(* CODESYS project plc_chalet_xplanar.library
   Title: CHALET_XPlanar
   Version: 4.3.3
   Placeholder: CHALET_XPlanar
   Company: Beckhoff CH

Project tree, tasks and I/O mapping:
  libraries: CHALET_BaseComponents, * (Beckhoff CH); CHALET_Nc, * (Beckhoff CH); Tc2_EtherCAT, * (Beckhoff Automation GmbH); Tc2_Math, * (Beckhoff Automation GmbH); Tc2_Standard, * (Beckhoff Automation GmbH); Tc2_System, * (Beckhoff Automation GmbH); Tc2_Utilities, * (Beckhoff Automation GmbH); Tc3_EventLogger, * (Beckhoff Automation GmbH); Tc3_Mc3Definitions, * (Beckhoff Automation GmbH); Tc3_Mc3PlanarMotion, * (Beckhoff Automation GmbH); Tc3_Module, * (Beckhoff Automation GmbH); Tc3_Physics, * (Beckhoff Automation GmbH); Tc3_XPlanarUtility, * (Beckhoff Automation GmbH & Co. KG)
  COMPONENTs/
    Environment/
      function block FB_XP_Environment [ST]: AddToGroup, RemoveFromGroup, Clear, Configure, FB_init, Feedback, Initialize, Mapped, OID, PlanarEnvironment, Update, UtilityEnvirement
      interface I_XP_Environment: AddToGroup, Clear, Configure, Feedback, Initialize, Mapped, OID, PlanarEnvironment, RemoveFromGroup, Update, UtilityEnvirement
    Feedback/
      function block FB_XP_Feedback [ST]: ClearObjectInfo, ObjectInfo
      interface I_XP_Feedback: ObjectInfo
    Group/
      function block FB_XP_Group [ST]: AddEnvironment, AddMover, AddTrack, Disable, Enable, FB_init, Feedback, Initialize, Mapped, OID, PlanarGroup, Reset, Update
      interface I_XP_Group: AddEnvironment, AddMover, AddTrack, Disable, Enable, Feedback, Initialize, Mapped, OID, PlanarGroup, Reset, Update
    Mover/
      ProductData/
        function block FB_XP_ProductData [ST]: LinkedMover, LinkToMover
        interface I_XP_ProductData: LinkedMover, LinkToMover
      function block FB_XP_Mover [ST]: DynConstraint, SetDynConstraint_A, SetDynConstraint_B, SetDynConstraint_C, SetDynConstraint_Path, SetDynConstraint_X, SetDynConstraint_Y, SetDynConstraint_Z, AxisExtSetpointA, AxisExtSetpointB, AxisExtSetpointC, AxisExtSetpointX, AxisExtSetpointY, AxisExtSetpointZ, StartExternalSetpoint, StopExternalSetpoint, UpdateExternalSetpoint, AddToGroup, RemoveFromGroup, Halt, MoveA, MoveB, MoveC, MoveXY, MoveZ, Disable, Enable, Reset, CommandMode, LagDistanceXY, PositionAct, PositionSet, CurrentTrack, DistToTrack, JoinTrack, LastCmdTargedGap, LastCmdTargedPosition, LastCmdTargedTrack, MoveOnTrack, MoveOnTrack_ShortestWay, MoveOnTrackToStation, ParentStation, PositionOnTrack, TargetStation, TcIoXPlanarMover, UtilityMover, DistToParentStation, FB_init, Feedback, Initialize, Mapped, Mode, OID, PlanarMover, Prepare, ProductData, Route, Update
      interface I_XP_Mover: AddToGroup, RemoveFromGroup, Halt, MoveA, MoveB, MoveC, MoveXY, MoveZ, Disable, Enable, Reset, CurrentTrack, DistToTrack, JoinTrack, LastCmdTargedGap, LastCmdTargedPosition, LastCmdTargedTrack, MoveOnTrack, MoveOnTrack_ShortestWay, MoveOnTrackToStation, ParentStation, PositionOnTrack, TargetStation, TcIoXPlanarMover, UtilityMover, DistToParentStation, Feedback, Mapped, Mode, OID, PlanarMover, Route
      interface I_XP_Mover_PLC: DynConstraint, SetDynConstraint_A, SetDynConstraint_B, SetDynConstraint_C, SetDynConstraint_Path, SetDynConstraint_X, SetDynConstraint_Y, SetDynConstraint_Z, AxisExtSetpointA, AxisExtSetpointB, AxisExtSetpointC, AxisExtSetpointX, AxisExtSetpointY, AxisExtSetpointZ, StartExternalSetpoint, StopExternalSetpoint, Halt, MoveA, MoveB, MoveC, MoveXY, MoveZ, CommandMode, LagDistanceXY, PositionAct, PositionSet, CurrentTrack, LastCmdTargedGap, LastCmdTargedPosition, LastCmdTargedTrack, ParentStation, PositionOnTrack, TargetStation, TcIoXPlanarMover, UtilityMover, DistToParentStation, Feedback, LUID, Mapped, OID, PlanarMover, ProductData
    Optional/
      Casting/
        function ToXpMover [ST]
        function ToXpStation [ST]
        function ToXpTrack [ST]
      Trigger/
        function block FB_XP_Trigger [ST]: AccocietedTrack, FB_init, HR, Initialize, ListOfMoversToCheck, MoverAtTrigger, MoverDetected, PositionOnTrack, Prepare, TimeStamp, TriggerDirection, Update
        interface I_XP_Trigger: AccocietedTrack, HR, ListOfMoversToCheck, MoverAtTrigger, MoverDetected, PositionOnTrack, TimeStamp, TriggerDirection
      Zone/
        function block FB_XP_SoretedListOfMover [ST]: CtsMoversInZone, FB_init, Initialize, MoversInZone, Prepare, Update
        interface I_XP_Zone: CtsMoversInZone, MoversInZone
      function F_GetDistToPosModulo [ST]
      function F_InLimitTest [ST]
      function block FB_XP_Path [ST]: DistanceToDestiantion, Length, LUID, PointerToThis, StationDestination, StationStart, TracksUsed
      interface I_XP_Path: DistanceToDestiantion, Length, PointerToThis, StationDestination, StationStart, TracksUsed
    Stationen/
      function block FB_XP_Station [ST]: CheckInvalideParameter, GetAccocietedTrack, GetDecisionDistance, GetPathsAhead, GetPathsBehind, GetPosOnTrack, GetStationAhead, GetStationBehinde, SetTrackObjName, Configure, CtsEmptySpaceInQueue, CtsMoversInQueue, MoverQueueSize, MoversInPlace, MoversInQueue, ReadyToRecvMovers, SendMoversToStation, SuppressDynamicsChange, TargetGroupe, TargetPosMonitoringTime, TargetPosWindow, ProcessSimulationActive, Simulation, SimulationMode, AccocietedTrack, AddMoverToQueue, AssignedMovers, DeleteMoversQueue, FB_exit, FB_init, Feedback, Filter, Initialize, MoverGapAtExit, MoverVelocityAtExit, OID, PathsAhead, PathsBehinde, PositionOnTrack, PositionOnTrackXY, PositionXY, Prepare, SearchNextBestStationByName, StationsAhead, StationsBehinde, Update
      interface I_XP_Station: AccocietedTrack, AddMoverToQueue, AssignedMovers, Configure, CtsEmptySpaceInQueue, DeleteMoversQueue, Filter, PathsAhead, PathsBehinde, PositionOnTrack, PositionOnTrackXY, PositionXY, ReadyToRecvMovers, SearchNextBestStationByName, SendMoversToStation, StationsAhead, StationsBehinde, TargetGroupe, Update
      interface I_XP_Station_PLC: CtsEmptySpaceInQueue, CtsMoversInQueue, LUID, MoverQueueSize, MoversInPlace, MoversInQueue, ReadyToRecvMovers, SendMoversToStation, TargetPosMonitoringTime, TargetPosWindow, ProcessSimulationActive, SimulationMode, AccocietedTrack, Feedback, Filter, MoverGapAtExit, PositionOnTrack, PositionOnTrackXY, PositionXY, StationsAhead, StationsBehinde, TargetGroupe
      data type ST_PathFinder_1
    System/
      function block FB_XP_System [ST]: JoiningStation, JoiningTrack, Disable, Disabled, Disabling, Enable, Enabled, Enabling, Initialize, Initialized, CheckTargetExists, Station, LinkEnvironment, LinkGroup, RegisterMover, RegisterStation, RegisterTrack, RegisterTrigger, RegisterZone, Enviroment, FB_init, Feedback, Movers, Stations, Tracks, Triggers, Update, XPlanarTaskAdsPort, Zones
      interface I_XP_System_PLC: CheckTargetExists, Disable, Disabled, Enable, Enabled, Enviroment, Feedback, Initialize, Initialized, Movers, Station, Stations, Tracks, Triggers, Update, Zones
      interface I_XP_System_Registration: LinkEnvironment, LinkGroup, RegisterMover, RegisterStation, RegisterTrack, RegisterTrigger, RegisterZone, Disabled, Enabled, Enviroment, Movers, Stations, Tracks, Triggers, XPlanarTaskAdsPort, Zones
    Track/
      function block FB_XP_Track [ST]: Configure, Configuring, Disable, Enable, AddToGroup, RemoveFromGroup, AddMover, ClosedLoop, CtsMoversOnTrack, FB_init, Feedback, Initialize, Length, Mapped, OID, PlanarTrack, Prepare, Reset, StationsOnTrack, TracksAhead, TracksBehinde, TracksEndAtThis, TracksStartFromThis, Update
      interface I_XP_Track: AddMover, AddToGroup, ClosedLoop, Configure, Configuring, CtsMoversOnTrack, Disable, Enable, Feedback, Length, OID, PlanarTrack, RemoveFromGroup, Reset, StationsOnTrack, TracksAhead, TracksBehinde, TracksEndAtThis, TracksStartFromThis
      interface I_XP_Track_PLC: CtsMoversOnTrack, Feedback, Length, Mapped, OID, PlanarTrack, StationsOnTrack, TracksAhead, TracksBehinde, TracksEndAtThis, TracksStartFromThis
  00000000-0000-0000-0000-000000000000|LICENSE.md
  LICENSE.md
  global variables XPlanarParameterlist
*)

// COMPONENTs/Stationen/ST_PathFinder_1
TYPE ST_PathFinder_1 :
STRUCT
	bTargetFound : BOOL; // Targed Station found on this path. No information about ready or not	
	fDistToTarged : LREAL := CHALET_BaseComponents.GVL_Datatypes.cMaxLreal;;
	ipBestStation : I_XP_Station; //to get to your destination, this would be the best station that can be reached directly and has space for at least 1 mover in the queue. Does not necessarily have to be the destination station
	ipRouteToParent : I_CH_LIST;
END_STRUCT
END_TYPE

// XPlanarParameterlist
{attribute 'qualified_only'}
VAR_GLOBAL CONSTANT 
	(*Minimum gap center to center on track [mm] *)
	F_MOVER_MINIMUM_GAP_ON_TRACK : LREAL := 100.0;
	
	(*During enabling the Movers use this gap [mm] *)
	F_GAP_STARTUP : LREAL := 150.0;
	
	(*Add envirement to groupe during enabling *)
	B_ADD_ENVIROMENT_TO_GROUP: BOOL := TRUE;	
		
	(*Pathfinder max recursion search depth in stations*)
	N_MAX_SEARCH_DEPTH: UINT := 50;
	
	(*The movers are only sent to the next free station on the way to the destination. 
	The distance in mm can be specified here to indicate how much further away the new move command can already be sent.  *)
	F_DIST_SET_NEW_MOVE_CMD_BEFORE_REACHING_PARENT_STATION : LREAL := 100.0;
	
	(*max tracks after a track switch *)
	N_MAX_STATIONS_AHEAD_OR_BEHIND : UINT := 10;	
	
	//Velocity during enabling move on track. 0=Default
	F_ENABLING_ON_TRACK_VELOCITY	: LREAL := 0;
	
	//Acc-/Deceleration during enabling move on track. 0=Default
	F_ENABLING_ON_TRACK_ACC_DEC		: LREAL := 0;
		
END_VAR

// COMPONENTs/Environment/FB_XP_Environment
{attribute 'no_explicit_call' := 'Do not call the body - Stick to OOP'}
(* XPlanar Environment - 1 per associated XPlanar 
	The Planar environment is a software object that represents the two-dimensional XPlanar stator surface. Together with Planar movers in a group, 
	it prevents collisions of the movers with the edge of the surface. *)
FUNCTION_BLOCK FB_XP_Environment EXTENDS FB_CH_Object IMPLEMENTS I_XP_Environment
VAR
	//Link to Planar-Environment object
	fbEnvironment : MC_PlanarEnvironment;
	fbUtilityEnvirement : FB_TcIoXPlanarEnvironment;
	
	{attribute 'hide'}  
	bInitDone :BOOL := FALSE;
	{attribute 'hide'}
	iXpSystem : I_XP_System_Registration;
	{attribute 'hide'}               	
	fbFeedback 			: FB_XP_Feedback;
	{attribute 'hide'}                   	
	eActiveCommand 		: CHALET_Nc.E_NcAxisCommands := CHALET_Nc.E_NcAxisCommands.None;
END_VAR


// Planar-Feedback objects
VAR
	{attribute 'hide'} 
	fbFeedbackAddToGrp : MC_PlanarFeedback;
	{attribute 'hide'} 
	fbFeedbackRmvFromGrp : MC_PlanarFeedback;
	{attribute 'hide'} 
	fbFeedbackConfigure : MC_PlanarFeedback;
	{attribute 'hide'} 
	fbFeedbackClear : MC_PlanarFeedback;
END_VAR

METHOD AddToGroup : HRESULT
VAR_INPUT
	iGroup : I_XP_Group;
END_VAR
IF NOT THIS^.fbFeedback.Busy THEN
	THIS^.eActiveCommand 				:= CHALET_NC.E_NcAxisCommands.AddToGroupe;
	THIS^.fbFeedback.LastCommandAccepted:= TRUE;		
	THIS^.fbFeedback.Busy 				:= TRUE;
	
	iGroup.AddEnvironment(THIS^.fbEnvironment, THIS^.fbFeedbackAddToGrp);
	AddToGroup := S_OK;
ELSE
	AddToGroup := S_FALSE;
	THIS^.fbFeedback.LastCommandAccepted:= FALSE;	
END_IF
END_METHOD

METHOD RemoveFromGroup : HRESULT
IF NOT THIS^.fbFeedback.Busy THEN
	THIS^.eActiveCommand 				:= CHALET_NC.E_NcAxisCommands.RemoveFromGroupe;
	THIS^.fbFeedback.LastCommandAccepted:= TRUE;		
	THIS^.fbFeedback.Busy 				:= TRUE;
	
	THIS^.fbEnvironment.RemoveFromGroup(THIS^.fbFeedbackRmvFromGrp);
	RemoveFromGroup := S_OK;
ELSE
	RemoveFromGroup := S_FALSE;
	THIS^.fbFeedback.LastCommandAccepted:= FALSE;	
END_IF
END_METHOD

METHOD Clear : HRESULT
THIS^.eActiveCommand 				:= CHALET_NC.E_NcAxisCommands.Clear;
THIS^.fbFeedback.LastCommandAccepted:= TRUE;		
THIS^.fbFeedback.Busy 				:= TRUE;

THIS^.fbEnvironment.Clear(commandFeedback:=THIS^.fbFeedbackClear);
Clear := S_OK;
END_METHOD

METHOD Configure : HRESULT
THIS^.eActiveCommand 				:= CHALET_NC.E_NcAxisCommands.Configure;
THIS^.fbFeedback.LastCommandAccepted:= TRUE;		
THIS^.fbFeedback.Busy 				:= TRUE;

THIS^.fbEnvironment.CreateBoundary(commandFeedback:=THIS^.fbFeedbackConfigure);
Configure := S_OK;
END_METHOD

METHOD FB_init : BOOL
VAR_INPUT
	bInitRetains : BOOL; // if TRUE, the retain variables are initialized (warm start / cold start)
	bInCopyCode : BOOL;  // if TRUE, the instance afterwards gets moved into the copy code (online change)
	
	ipSystem : I_CH_Object;
END_VAR
VAR_INST
	{attribute 'hide'}
	bFBInitCalledOnce : BOOL; //Do the following code once during start up and not during onlinechange
END_VAR
//Do the following code once during start up and not during onlinechange
IF NOT bFBInitCalledOnce THEN 
	
	(* Register to the Xplanar System
	   1. Test if the interface exists
	   2. Test if the object implements a "System for Mover" interface 
	*)
	IF ipSystem <> 0 AND_THEN __QUERYINTERFACE(ipSystem,THIS^.iXpSystem) THEN
		THIS^.iXpSystem.LinkEnvironment(THIS^);
	END_IF
	
	
END_IF

bFBInitCalledOnce := TRUE;
END_METHOD

{attribute 'monitoring':='call'}
PROPERTY Feedback : I_XP_Feedback
GET
Feedback := THIS^.fbFeedback;
END_GET
END_PROPERTY

METHOD Initialize : HRESULT
VAR
	stVarInfo : __SYSTEM.VAR_INFO;
END_VAR
VAR_INST
	//This error cannot be reset. Requires a reset cold
	{attribute 'hide'}	
	fbInitError : FB_TcAlarm;
END_VAR
// Check if link to envirement is mapped
IF NOT THIS^.Mapped THEN
	IF NOT fbInitError.bRaised THEN 
		//This error cannot be reset. Requires a reset cold
		fbInitError.CreateEx(stEventEntry:=TC_EVENTS.CHALET_XPlanar_Events.VariableLinkMissing, ipSourceInfo := THIS^.fbSourceInfo, bWithConfirmation := FALSE);
		stVarInfo := __VARINFO(fbEnvironment);
		fbInitError.ipArguments.AddString(stVarInfo.Symbol);
		fbInitError.Raise(0);
	END_IF
	Initialize := E_FAIL;
	RETURN;
END_IF



IF NOT bInitDone THEN
	//Busy
	Initialize := S_PENDING;
	
	IF fbUtilityEnvirement.Init(bExecute := TRUE) THEN
		fbUtilityEnvirement.Init(bExecute := FALSE);
		bInitDone := TRUE;
	END_IF
	
	
ELSE	
	//Done
	Initialize := S_OK;
END_IF



THIS^.fbFeedback.ActiveCommand 		:= TO_STRING(CHALET_NC.E_NcAxisCommands.Initialize);
THIS^.eActiveCommand 				:= CHALET_NC.E_NcAxisCommands.Initialize;
THIS^.fbFeedback.LastCommandAccepted:= TRUE;	
//Set done or keep in busy state	
THIS^.fbFeedback.HR := Initialize;
END_METHOD

{attribute 'monitoring':='call'}
PROPERTY Mapped : BOOL //Project is mapped to MC (McToPlc and PlcToMc)
GET
VAR
	bMcToPlcNotMapped 	: BOOL;
END_VAR
bMcToPlcNotMapped := F_GetMappingStatus(ADR(THIS^.fbEnvironment.MCTOPLC_STD), SIZEOF(THIS^.fbEnvironment.MCTOPLC_STD)) <> EPlcMappingStatus.MS_Mapped;

Mapped := NOT bMcToPlcNotMapped;
END_GET
END_PROPERTY

{attribute 'monitoring':='call'}
//Unique object ID
PROPERTY OID : OTCID
GET
OID := THIS^.fbEnvironment.MCTOPLC_STD.EnvironmentOID;
END_GET
END_PROPERTY

{attribute 'monitoring':='call'}
PROPERTY PlanarEnvironment : REFERENCE TO MC_PlanarEnvironment
GET
PlanarEnvironment ref= THIS^.fbEnvironment;
END_GET
END_PROPERTY

METHOD PUBLIC Update : HRESULT
VAR_INPUT
END_VAR



// ********************** Set feedback depending on active command *******************************
IF THIS^.eActiveCommand <> E_NcAxisCommands.None THEN
	fbFeedback.ActiveCommand 	:= TO_STRING(THIS^.eActiveCommand);	
END_IF

CASE THIS^.eActiveCommand OF
	E_NcAxisCommands.None: 
		//Display if a Mover Error is active during no command is active
		IF THIS^.fbEnvironment.Error AND NOT fbFeedback.Error THEN 
			fbFeedback.ErrorId 			:= THIS^.fbEnvironment.ErrorID;
			fbFeedback.ActiveCommand 	:= TO_STRING(E_NcAxisCommands.None);	
			fbFeedback.ClearObjectInfo();
		END_IF

	E_NcAxisCommands.Initialize:
		fbFeedback.Busy 			:= NOT THIS^.bInitDone;
		fbFeedback.Done 			:= THIS^.bInitDone;
		fbFeedback.ErrorId 			:= 0;
		fbFeedback.ClearObjectInfo();
		                                                       			                        	
	E_NcAxisCommands.Clear:     	
		fbFeedback.Busy 			:= fbFeedbackClear.Busy;
		fbFeedback.Done 			:= fbFeedbackClear.Done;
		fbFeedback.ErrorId 			:= fbFeedbackClear.ErrorID;
        fbFeedback.ObjectInfo		:= fbFeedbackClear.objectInfo;
           			                        	
	E_NcAxisCommands.Configure:     	
		fbFeedback.Busy 			:= fbFeedbackConfigure.Busy;
		fbFeedback.Done 			:= fbFeedbackConfigure.Done;
		fbFeedback.ErrorId 			:= fbFeedbackConfigure.ErrorID;
        fbFeedback.ObjectInfo		:= fbFeedbackConfigure.objectInfo;
                                      			                        	
	E_NcAxisCommands.AddToGroupe:     	
		fbFeedback.Busy 			:= fbFeedbackAddToGrp.Busy;
		fbFeedback.Done 			:= fbFeedbackAddToGrp.Done;
		fbFeedback.ErrorId 			:= fbFeedbackAddToGrp.ErrorID;
        fbFeedback.ObjectInfo		:= fbFeedbackAddToGrp.objectInfo;
                                      			                        	
	E_NcAxisCommands.RemoveFromGroupe:     	
		fbFeedback.Busy 			:= fbFeedbackRmvFromGrp.Busy;
		fbFeedback.Done 			:= fbFeedbackRmvFromGrp.Done;
		fbFeedback.ErrorId 			:= fbFeedbackRmvFromGrp.ErrorID;
        fbFeedback.ObjectInfo		:= fbFeedbackRmvFromGrp.objectInfo;
                                		
	ELSE//External command in subclass
		;
END_CASE


// **********************  Stop to execute commands on .done or .error ***************************
IF fbFeedback.Done OR THIS^.fbFeedback.Error THEN
	eActiveCommand 				:= E_NcAxisCommands.None;
END_IF

//Update xplanar object
THIS^.fbEnvironment.Update();

//Update feedback object
fbFeedbackConfigure.Update(); 
fbFeedbackClear.Update(); 
fbFeedbackAddToGrp.Update(); 
fbFeedbackRmvFromGrp.Update();
END_METHOD

{attribute 'monitoring':='call'}
PROPERTY UtilityEnvirement : Tc3_XPlanarUtility.I_Environment
GET
UtilityEnvirement := fbUtilityEnvirement;
END_GET
END_PROPERTY

END_FUNCTION_BLOCK

// COMPONENTs/Environment/I_XP_Environment
INTERFACE I_XP_Environment  EXTENDS __SYSTEM.IQueryInterface, I_CH_Object

METHOD AddToGroup : HRESULT
VAR_INPUT
	iGroup : I_XP_Group;
END_VAR
END_METHOD

METHOD Clear : HRESULT
END_METHOD

METHOD Configure : HRESULT
VAR_INPUT
END_VAR
END_METHOD

{attribute 'monitoring':='call'}
PROPERTY Feedback : I_XP_Feedback
GET
END_GET
END_PROPERTY

METHOD Initialize : HRESULT
END_METHOD

{attribute 'monitoring':='call'}
PROPERTY Mapped : BOOL //Project is mapped to MC (McToPlc and PlcToMc)
GET
END_GET
END_PROPERTY

{attribute 'monitoring':='call'}
//Unique object ID
PROPERTY OID : OTCID
GET
END_GET
END_PROPERTY

{attribute 'monitoring':='call'}
PROPERTY PlanarEnvironment : REFERENCE TO MC_PlanarEnvironment
GET
END_GET
END_PROPERTY

METHOD RemoveFromGroup : HRESULT
END_METHOD

METHOD PUBLIC Update : HRESULT
VAR_INPUT
END_VAR
END_METHOD

{attribute 'monitoring':='call'}
PROPERTY UtilityEnvirement : Tc3_XPlanarUtility.I_Environment
GET
END_GET
END_PROPERTY

END_INTERFACE

// COMPONENTs/Group/I_XP_Group
INTERFACE I_XP_Group  EXTENDS __SYSTEM.IQueryInterface, I_CH_Object

METHOD AddEnvironment : HRESULT
VAR_INPUT
	refEnvironment : REFERENCE TO MC_PlanarEnvironment;
	refFeedback : REFERENCE TO MC_PlanarFeedback;
END_VAR
END_METHOD

METHOD AddMover : HRESULT
VAR_INPUT
	refMover : REFERENCE TO MC_PlanarMover;
	refFeedback : REFERENCE TO MC_PlanarFeedback;
END_VAR
END_METHOD

METHOD AddTrack : HRESULT
VAR_INPUT
	refTrack : REFERENCE TO MC_PlanarTrack;
	refFeedback : REFERENCE TO MC_PlanarFeedback;
END_VAR
END_METHOD

METHOD Disable : HRESULT
VAR_INPUT
END_VAR
END_METHOD

METHOD Enable : HRESULT
VAR_INPUT
END_VAR
END_METHOD

{attribute 'OPC.UA.DA.Property' := '1'}
{attribute 'monitoring':='call'}
PROPERTY Feedback : I_XP_Feedback
GET
END_GET
END_PROPERTY

METHOD Initialize : HRESULT
VAR_INPUT
END_VAR
END_METHOD

{attribute 'monitoring':='call'}
PROPERTY Mapped : BOOL //Project is mapped to MC (McToPlc and PlcToMc)
GET
END_GET
END_PROPERTY

{attribute 'monitoring':='call'}
//Unique object ID
PROPERTY OID : OTCID
GET
END_GET
END_PROPERTY

{attribute 'monitoring':='call'}
PROPERTY PlanarGroup : REFERENCE TO MC_PlanarGroup
GET
END_GET
END_PROPERTY

METHOD Reset : HRESULT
VAR_INPUT
END_VAR
END_METHOD

METHOD PUBLIC Update : HRESULT
VAR_INPUT
END_VAR
END_METHOD

END_INTERFACE

// COMPONENTs/Feedback/I_XP_Feedback
INTERFACE I_XP_Feedback EXTENDS CHALET_BaseComponents.I_CH_Feedback

{attribute 'monitoring':='call'}
(* Indicates which object one would collide with. *)
PROPERTY ObjectInfo : REFERENCE TO PlanarObjectInfo
GET
END_GET
END_PROPERTY

END_INTERFACE

// COMPONENTs/System/I_XP_System_Registration
INTERFACE I_XP_System_Registration EXTENDS __SYSTEM.IQueryInterface

METHOD LinkEnvironment : HRESULT
VAR_INPUT
	ipEnvironment : I_CH_Object;
END_VAR
END_METHOD

METHOD LinkGroup : HRESULT
VAR_INPUT
	ipGroup : I_CH_Object;
END_VAR
END_METHOD

METHOD RegisterMover : HRESULT
VAR_INPUT
	ipMover : I_CH_Object;
END_VAR
END_METHOD

METHOD RegisterStation : HRESULT
VAR_INPUT
	ipStation : I_CH_Object;
END_VAR
END_METHOD

METHOD RegisterTrack : HRESULT
VAR_INPUT
	ipTrack : I_CH_Object;
END_VAR
END_METHOD

METHOD RegisterTrigger : HRESULT
VAR_INPUT
	ipTrigger	: CHALET_BaseComponents.I_CH_Object;
END_VAR
END_METHOD

METHOD RegisterZone : HRESULT
VAR_INPUT
	ipZone	: CHALET_BaseComponents.I_CH_Object;
END_VAR
END_METHOD

{attribute 'monitoring':='call'}
PROPERTY Disabled : BOOL
GET
END_GET
END_PROPERTY

{attribute 'monitoring':='call'}
PROPERTY Enabled : BOOL
GET
END_GET
END_PROPERTY

{attribute 'monitoring':='call'}
PROPERTY Enviroment : I_XP_Environment
GET
END_GET
END_PROPERTY

{attribute 'monitoring':='call'}
PROPERTY Movers : CHALET_BaseComponents.I_CH_LIST
GET
END_GET
END_PROPERTY

{attribute 'monitoring':='call'}
PROPERTY Stations : CHALET_BaseComponents.I_CH_LIST
GET
END_GET
END_PROPERTY

{attribute 'monitoring':='call'}
PROPERTY Tracks : CHALET_BaseComponents.I_CH_LIST
GET
END_GET
END_PROPERTY

{attribute 'monitoring':='call'}
PROPERTY Triggers : CHALET_BaseComponents.I_CH_LIST
GET
END_GET
END_PROPERTY

{attribute 'monitoring':='call'}
PROPERTY XPlanarTaskAdsPort : UINT
GET
END_GET
END_PROPERTY

{attribute 'monitoring':='call'}
PROPERTY Zones : CHALET_BaseComponents.I_CH_LIST
GET
END_GET
END_PROPERTY

END_INTERFACE

// COMPONENTs/Feedback/FB_XP_Feedback
{attribute 'no_explicit_call' := 'Do not call the body - Stick to OOP'}
FUNCTION_BLOCK FB_XP_Feedback EXTENDS CHALET_BaseComponents.FB_CH_Feedback IMPLEMENTS I_XP_Feedback
VAR_INPUT
END_VAR
VAR_OUTPUT
END_VAR
VAR
	(* Indicates which object one would collide with. *)
	{attribute 'hide'}
	_objectInfo : PlanarObjectInfo;
END_VAR

METHOD ClearObjectInfo : BOOL
VAR_INPUT
END_VAR
THIS^._ObjectInfo.Id := 0;
THIS^._ObjectInfo.ObjectType := EPlanarObjectType.None;
END_METHOD

{attribute 'monitoring':='call'}
(* Indicates which object one would collide with. *)
PROPERTY ObjectInfo : REFERENCE TO PlanarObjectInfo
GET
objectInfo REF= THIS^._objectInfo;
END_GET
END_PROPERTY

END_FUNCTION_BLOCK

// COMPONENTs/Group/FB_XP_Group
{attribute 'no_explicit_call' := 'Do not call the body - Stick to OOP'}
(* XPlanar Collision Avoidance Groupe - 1 per associated XPlanar 
	The Planar group is a software object that prevents collisions between Planar movers as well as collisions of Planar movers with the boundary of 
	the stator area on the two-dimensional XPlanar stator area. To do this, the 2D areas of all objects in the group are blocked. When a motion command 
	is transferred to a mover, the required area is requested from the Planar group and the motion command is rejected if this area would collide 
	with already reserved areas. If the motion command can be executed, the area is added to the set of reserved area and blocked accordingly. *)
FUNCTION_BLOCK FB_XP_Group EXTENDS FB_CH_Object IMPLEMENTS I_XP_Group
VAR
	//Link to Planar-Group object
	fbGroup : MC_PlanarGroup;
		
	{attribute 'hide'}  
	bInitDone :BOOL := FALSE;
	{attribute 'hide'}
	iXpSystem : I_XP_System_Registration;
	{attribute 'hide'}               	
	fbFeedback 			: FB_XP_Feedback;
	{attribute 'hide'}                   	
	eActiveCommand 		: CHALET_Nc.E_NcAxisCommands := CHALET_Nc.E_NcAxisCommands.None;

END_VAR


// Planar-Feedback objects
VAR
	{attribute 'hide'} 
	fbFeedbackDisable : MC_PlanarFeedback;
	{attribute 'hide'} 
	fbFeedbackEnable : MC_PlanarFeedback;
	{attribute 'hide'} 
	fbFeedbackReset : MC_PlanarFeedback;
END_VAR

METHOD AddEnvironment : HRESULT
VAR_INPUT
	refEnvironment : REFERENCE TO MC_PlanarEnvironment;
	refFeedback : REFERENCE TO MC_PlanarFeedback;
END_VAR
refEnvironment.AddToGroup(refFeedback, fbGroup);
END_METHOD

METHOD AddMover : HRESULT
VAR_INPUT
	refMover : REFERENCE TO MC_PlanarMover;
	refFeedback : REFERENCE TO MC_PlanarFeedback;
END_VAR
refMover.AddToGroup(refFeedback, fbGroup);
END_METHOD

METHOD AddTrack : HRESULT
VAR_INPUT
	refTrack : REFERENCE TO MC_PlanarTrack;
	refFeedback : REFERENCE TO MC_PlanarFeedback;
END_VAR
refTrack.AddToGroup(refFeedback, fbGroup);
END_METHOD

METHOD Disable : HRESULT
VAR_INPUT
END_VAR
THIS^.eActiveCommand 				:= CHALET_NC.E_NcAxisCommands.Disable;
THIS^.fbFeedback.LastCommandAccepted:= TRUE;		
THIS^.fbFeedback.Busy 				:= TRUE;

THIS^.fbGroup.Disable(fbFeedbackDisable);

Disable := S_OK;
END_METHOD

METHOD Enable : HRESULT
VAR_INPUT
END_VAR
IF NOT THIS^.fbFeedback.Busy THEN
	THIS^.eActiveCommand 				:= CHALET_NC.E_NcAxisCommands.Enable;
	THIS^.fbFeedback.LastCommandAccepted:= TRUE;		
	THIS^.fbFeedback.Busy 				:= TRUE;

	THIS^.fbGroup.Enable(fbFeedbackEnable);
	Enable := S_OK;
ELSE
	Enable := S_FALSE;
	THIS^.fbFeedback.LastCommandAccepted:= FALSE;	
END_IF
END_METHOD

METHOD FB_init : BOOL
VAR_INPUT
	bInitRetains : BOOL; // if TRUE, the retain variables are initialized (warm start / cold start)
	bInCopyCode : BOOL;  // if TRUE, the instance afterwards gets moved into the copy code (online change)
	
	ipSystem : I_CH_Object;
END_VAR
VAR_INST
	{attribute 'hide'}
	bFBInitCalledOnce : BOOL; //Do the following code once during start up and not during onlinechange
END_VAR
//Do the following code once during start up and not during onlinechange
IF NOT bFBInitCalledOnce THEN 
	

	(* Register to the Xplanar System
	   1. Test if the interface exists
	   2. Test if the object implements a "System for Mover" interface 
	*)
	IF ipSystem <> 0 AND_THEN __QUERYINTERFACE(ipSystem,THIS^.iXpSystem) THEN
		THIS^.iXpSystem.LinkGroup(THIS^);
	END_IF
	
	
END_IF

bFBInitCalledOnce := TRUE;
END_METHOD

{attribute 'monitoring':='call'}
PROPERTY Feedback : I_XP_Feedback
GET
Feedback := THIS^.fbFeedback;
END_GET
END_PROPERTY

METHOD Initialize : HRESULT
VAR_INPUT
END_VAR
VAR
	stVarInfo : __SYSTEM.VAR_INFO;
END_VAR
VAR_INST
	//This error cannot be reset. Requires a reset cold
	{attribute 'hide'}	
	fbInitError : FB_TcAlarm;
END_VAR
// Check if link to MC-Mover is mapped
IF NOT THIS^.Mapped THEN
	IF NOT fbInitError.bRaised THEN 
		//This error cannot be reset. Requires a reset cold
		fbInitError.CreateEx(stEventEntry:=TC_EVENTS.CHALET_XPlanar_Events.VariableLinkMissing, ipSourceInfo := THIS^.fbSourceInfo, bWithConfirmation := FALSE);
		stVarInfo := __VARINFO(fbGroup);
		fbInitError.ipArguments.AddString(stVarInfo.Symbol);
		fbInitError.Raise(0);
	END_IF
	Initialize := E_FAIL;
	RETURN;
END_IF


IF NOT bInitDone THEN
	//Busy
	Initialize := S_PENDING;

	bInitDone := TRUE;	
	
ELSE	
	//Done
	Initialize := S_OK;	
END_IF



THIS^.fbFeedback.ActiveCommand 		:= TO_STRING(CHALET_NC.E_NcAxisCommands.Initialize);
THIS^.eActiveCommand 				:= CHALET_NC.E_NcAxisCommands.Initialize;
THIS^.fbFeedback.LastCommandAccepted:= TRUE;	
//Set done or keep in busy state	
THIS^.fbFeedback.HR := Initialize;
END_METHOD

{attribute 'monitoring':='call'}
PROPERTY Mapped : BOOL //Project is mapped to MC (McToPlc and PlcToMc)
GET
VAR
	bMcToPlcNotMapped 	: BOOL;
END_VAR
bMcToPlcNotMapped := F_GetMappingStatus(ADR(THIS^.fbGroup.MCTOPLC_STD), SIZEOF(THIS^.fbGroup.MCTOPLC_STD)) <> EPlcMappingStatus.MS_Mapped;

Mapped := NOT bMcToPlcNotMapped;
END_GET
END_PROPERTY

{attribute 'monitoring':='call'}
//Unique object ID
PROPERTY OID : OTCID
GET
OID := THIS^.fbGroup.MCTOPLC_STD.GroupOID;
END_GET
END_PROPERTY

{attribute 'monitoring':='call'}
PROPERTY PlanarGroup : REFERENCE TO MC_PlanarGroup
GET
PlanarGroup ref= THIS^.fbGroup;
END_GET
END_PROPERTY

METHOD Reset : HRESULT
VAR_INPUT
END_VAR
IF NOT THIS^.fbFeedback.Busy THEN
	THIS^.eActiveCommand 				:= CHALET_NC.E_NcAxisCommands.Reset;
	THIS^.fbFeedback.LastCommandAccepted:= TRUE;		
	THIS^.fbFeedback.Busy 				:= TRUE;

	THIS^.fbGroup.Reset(fbFeedbackReset);
	Reset := S_OK;
ELSE
	Reset := S_FALSE;
	THIS^.fbFeedback.LastCommandAccepted:= FALSE;		
END_IF
END_METHOD

METHOD PUBLIC Update : HRESULT
VAR_INPUT
END_VAR



// ********************** Set feedback depending on active command *******************************
IF THIS^.eActiveCommand <> E_NcAxisCommands.None THEN
	fbFeedback.ActiveCommand 	:= TO_STRING(THIS^.eActiveCommand);	
END_IF

CASE THIS^.eActiveCommand OF
	E_NcAxisCommands.None: 
		//Display if a Mover Error is active during no command is active
		IF THIS^.fbGroup.Error AND NOT fbFeedback.Error THEN 
			fbFeedback.ErrorId 			:= THIS^.fbGroup.ErrorID;
			fbFeedback.ActiveCommand 	:= TO_STRING(E_NcAxisCommands.None);	
			fbFeedback.ClearObjectInfo();
		END_IF

	E_NcAxisCommands.Initialize:
		fbFeedback.Busy 			:= NOT THIS^.bInitDone;
		fbFeedback.Done 			:= THIS^.bInitDone;
		fbFeedback.ErrorId 			:= 0;
		fbFeedback.ClearObjectInfo();
		                        	
	E_NcAxisCommands.Enable:     	
		fbFeedback.Busy 			:= fbFeedbackEnable.Busy;
		fbFeedback.Done 			:= fbFeedbackEnable.Done;
		fbFeedback.ErrorId 			:= fbFeedbackEnable.ErrorID;
        fbFeedback.ObjectInfo		:= fbFeedbackEnable.objectInfo;
                                			                        	
	E_NcAxisCommands.Disable:     	
		fbFeedback.Busy 			:= fbFeedbackDisable.Busy;
		fbFeedback.Done 			:= fbFeedbackDisable.Done;
		fbFeedback.ErrorId 			:= fbFeedbackDisable.ErrorID;
        fbFeedback.ObjectInfo		:= fbFeedbackDisable.objectInfo;
                                			                        	
	E_NcAxisCommands.Reset:     	
		fbFeedback.Busy 			:= fbFeedbackReset.Busy;
		fbFeedback.Done 			:= fbFeedbackReset.Done;
		fbFeedback.ErrorId 			:= fbFeedbackReset.ErrorID;
        fbFeedback.ObjectInfo		:= fbFeedbackReset.objectInfo;
                                		
	ELSE//External command in subclass
		;
END_CASE


// **********************  Stop to execute commands on .done or .error ***************************
IF fbFeedback.Done OR THIS^.fbFeedback.Error THEN
	eActiveCommand 				:= E_NcAxisCommands.None;
END_IF

//Update xplanar object
THIS^.fbGroup.Update();

//Update feedback object
fbFeedbackEnable.Update(); 
fbFeedbackDisable.Update(); 
fbFeedbackReset.Update();
END_METHOD

END_FUNCTION_BLOCK

// COMPONENTs/Mover/ProductData/FB_XP_ProductData
FUNCTION_BLOCK FB_XP_ProductData EXTENDS FB_CH_Object IMPLEMENTS I_XP_ProductData
VAR
	{attribute 'hide'}
	ipMover : I_XP_Mover_PLC;
END_VAR

{attribute 'monitoring':='call'}
PROPERTY LinkedMover : I_XP_Mover_PLC
GET
LinkedMover := ipMover;
END_GET
END_PROPERTY

METHOD LinkToMover : BOOL //it is not necessary to call this method. This is already done internally
VAR_INPUT
	ipMoverPlc : I_XP_Mover_PLC;
END_VAR
THIS^.ipMover := ipMoverPlc;
END_METHOD

END_FUNCTION_BLOCK

// COMPONENTs/Mover/ProductData/I_XP_ProductData
INTERFACE I_XP_ProductData EXTENDS __SYSTEM.IQueryInterface

{attribute 'monitoring':='call'}
PROPERTY LinkedMover : I_XP_Mover_PLC
GET
END_GET
END_PROPERTY

METHOD LinkToMover : BOOL //it is not necessary to call this method. This is already done internally
VAR_INPUT
	ipMoverPlc : I_XP_Mover_PLC;
END_VAR
END_METHOD

END_INTERFACE

// COMPONENTs/Mover/I_XP_Mover_PLC
INTERFACE I_XP_Mover_PLC EXTENDS __SYSTEM.IQueryInterface

PROPERTY DynConstraint : REFERENCE TO DynamicConstraint_Container
GET
END_GET
END_PROPERTY

METHOD SetDynConstraint_A : BOOL //Dynamic constraints for individual coordinates.
VAR_INPUT
    V : MC_LREAL; //equivalent to data type LREAL + MC_DEFAULT, MC_MAXIMUM
    A : MC_LREAL; //equivalent to data type LREAL + MC_DEFAULT, MC_MAXIMUM
    D : MC_LREAL; //equivalent to data type LREAL + MC_DEFAULT, MC_MAXIMUM
    J : MC_LREAL; //equivalent to data type LREAL + MC_DEFAULT, MC_MAXIMUM
END_VAR
END_METHOD

METHOD SetDynConstraint_B : BOOL //Dynamic constraints for individual coordinates.
VAR_INPUT
    V : MC_LREAL; //equivalent to data type LREAL + MC_DEFAULT, MC_MAXIMUM
    A : MC_LREAL; //equivalent to data type LREAL + MC_DEFAULT, MC_MAXIMUM
    D : MC_LREAL; //equivalent to data type LREAL + MC_DEFAULT, MC_MAXIMUM
    J : MC_LREAL; //equivalent to data type LREAL + MC_DEFAULT, MC_MAXIMUM
END_VAR
END_METHOD

METHOD SetDynConstraint_C : BOOL //Dynamic constraints for individual coordinates.
VAR_INPUT
    V : MC_LREAL; //equivalent to data type LREAL + MC_DEFAULT, MC_MAXIMUM
    A : MC_LREAL; //equivalent to data type LREAL + MC_DEFAULT, MC_MAXIMUM
    D : MC_LREAL; //equivalent to data type LREAL + MC_DEFAULT, MC_MAXIMUM
    J : MC_LREAL; //equivalent to data type LREAL + MC_DEFAULT, MC_MAXIMUM
END_VAR
END_METHOD

METHOD SetDynConstraint_Path : BOOL //One dimensional dynamic constraint along the XY-components of a path, ignoring non-tangential effects.
VAR_INPUT
    V : MC_LREAL; //equivalent to data type LREAL + MC_DEFAULT, MC_MAXIMUM
    A : MC_LREAL; //equivalent to data type LREAL + MC_DEFAULT, MC_MAXIMUM
    D : MC_LREAL; //equivalent to data type LREAL + MC_DEFAULT, MC_MAXIMUM
    J : MC_LREAL; //equivalent to data type LREAL + MC_DEFAULT, MC_MAXIMUM
END_VAR
END_METHOD

METHOD SetDynConstraint_X : BOOL //Dynamic constraints for individual coordinates.
VAR_INPUT
    V : MC_LREAL; //equivalent to data type LREAL + MC_DEFAULT, MC_MAXIMUM
    A : MC_LREAL; //equivalent to data type LREAL + MC_DEFAULT, MC_MAXIMUM
    D : MC_LREAL; //equivalent to data type LREAL + MC_DEFAULT, MC_MAXIMUM
    J : MC_LREAL; //equivalent to data type LREAL + MC_DEFAULT, MC_MAXIMUM
END_VAR
END_METHOD

METHOD SetDynConstraint_Y : BOOL //Dynamic constraints for individual coordinates.
VAR_INPUT
    V : MC_LREAL; //equivalent to data type LREAL + MC_DEFAULT, MC_MAXIMUM
    A : MC_LREAL; //equivalent to data type LREAL + MC_DEFAULT, MC_MAXIMUM
    D : MC_LREAL; //equivalent to data type LREAL + MC_DEFAULT, MC_MAXIMUM
    J : MC_LREAL; //equivalent to data type LREAL + MC_DEFAULT, MC_MAXIMUM
END_VAR
END_METHOD

METHOD SetDynConstraint_Z : BOOL //Dynamic constraints for individual coordinates.
VAR_INPUT
    V : MC_LREAL; //equivalent to data type LREAL + MC_DEFAULT, MC_MAXIMUM
    A : MC_LREAL; //equivalent to data type LREAL + MC_DEFAULT, MC_MAXIMUM
    D : MC_LREAL; //equivalent to data type LREAL + MC_DEFAULT, MC_MAXIMUM
    J : MC_LREAL; //equivalent to data type LREAL + MC_DEFAULT, MC_MAXIMUM
END_VAR
END_METHOD

{attribute 'monitoring':='call'}
PROPERTY  AxisExtSetpointA : CHALET_Nc.I_NcAxis_PLC
GET
END_GET
END_PROPERTY

{attribute 'monitoring':='call'}
PROPERTY AxisExtSetpointB : CHALET_Nc.I_NcAxis_PLC
GET
END_GET
END_PROPERTY

{attribute 'monitoring':='call'}
PROPERTY AxisExtSetpointC : CHALET_Nc.I_NcAxis_PLC
GET
END_GET
END_PROPERTY

{attribute 'monitoring':='call'}
PROPERTY  AxisExtSetpointX : CHALET_Nc.I_NcAxis_PLC
GET
END_GET
END_PROPERTY

{attribute 'monitoring':='call'}
PROPERTY AxisExtSetpointY : CHALET_Nc.I_NcAxis_PLC
GET
END_GET
END_PROPERTY

{attribute 'monitoring':='call'}
PROPERTY AxisExtSetpointZ : CHALET_Nc.I_NcAxis_PLC
GET
END_GET
END_PROPERTY

METHOD StartExternalSetpoint : HRESULT
END_METHOD

METHOD StopExternalSetpoint : HRESULT
VAR_INPUT
END_VAR
END_METHOD

METHOD Halt : HRESULT
VAR_INPUT
END_VAR
END_METHOD

METHOD MoveA : HRESULT
VAR_INPUT
	fPosition : LREAL;
END_VAR
END_METHOD

METHOD MoveB : HRESULT
VAR_INPUT
	fPosition : LREAL;
END_VAR
END_METHOD

METHOD MoveC : HRESULT
VAR_INPUT
	fPosition : LREAL;
	
	(* Addition turns to move in modulo movement (positive or negative). *)
	additionalTurns : UDINT := 0;
	
	(* Direction in which the target is approached. *)
	direction : Tc3_Mc3Definitions.MC_DIRECTION := Tc3_Mc3Definitions.MC_DIRECTION.mcDirectionNonModulo;
END_VAR
END_METHOD

METHOD MoveXY : HRESULT
VAR_INPUT
	fPosition_X : LREAL;
	fPosition_Y : LREAL;
END_VAR
END_METHOD

METHOD MoveZ : HRESULT
VAR_INPUT
	fPosition : LREAL;
END_VAR
END_METHOD

{attribute 'monitoring':='call'}
(* Indicates the command mode of an enabled PlanarMover, i.e. how setpoints are currently produced. *)
PROPERTY CommandMode : MC_PLANAR_MOVER_COMMAND_MODE
GET
END_GET
END_PROPERTY

{attribute 'monitoring':='call'}
(* Retruns lentgh of hypotenuse of the x and y error. (>=0[mm]) *)
PROPERTY LagDistanceXY : LREAL
GET
END_GET
END_PROPERTY

{attribute 'monitoring':='call'}
(* Contains the information of the Planar Mover passed from MC to PLC. XYZABC [mm] *)
PROPERTY PositionAct : REFERENCE TO MoverVector
GET
END_GET
END_PROPERTY

{attribute 'monitoring':='call'}
(* Provides the current planar mover setpoint XYZABC [mm] *)
PROPERTY PositionSet : REFERENCE TO MoverVector
GET
END_GET
END_PROPERTY

{attribute 'monitoring':='call'}
PROPERTY CurrentTrack : I_XP_Track
GET
END_GET
END_PROPERTY

{attribute 'monitoring':='call'}
PROPERTY LastCmdTargedGap : LREAL
GET
END_GET
END_PROPERTY

{attribute 'monitoring':='call'}
PROPERTY LastCmdTargedPosition : LREAL
GET
END_GET
END_PROPERTY

{attribute 'monitoring':='call'}
PROPERTY LastCmdTargedTrack: I_XP_Track
GET
END_GET
END_PROPERTY

{attribute 'monitoring':='call'}
PROPERTY ParentStation : I_XP_Station
GET
END_GET
END_PROPERTY

{attribute 'monitoring':='call'}
PROPERTY PositionOnTrack : LREAL
GET
END_GET
END_PROPERTY

{attribute 'monitoring':='call'}
PROPERTY TargetStation : STRING
GET
END_GET
SET
END_SET
END_PROPERTY

{attribute 'monitoring':='call'}
PROPERTY TcIoXPlanarMover : Tc3_XPlanarUtility.I_TcIoXPlanarMover
GET
END_GET
END_PROPERTY

{attribute 'monitoring':='call'}
PROPERTY UtilityMover : Tc3_XPlanarUtility.I_McPlanarMover
GET
END_GET
END_PROPERTY

{attribute 'monitoring':='call'}
PROPERTY DistToParentStation : LREAL //Distance to the responsible parent station [mm]
GET
END_GET
END_PROPERTY

{attribute 'OPC.UA.DA.Property' := '1'}
{attribute 'monitoring':='call'}
PROPERTY Feedback : I_XP_Feedback
GET
END_GET
END_PROPERTY

{attribute 'monitoring':='call'}
PROPERTY LUID : STRING //Locally unique identifier
GET
END_GET
END_PROPERTY

{attribute 'monitoring':='call'}
PROPERTY Mapped : BOOL //Project is mapped to MC (McToPlc and PlcToMc)
GET
END_GET
END_PROPERTY

{attribute 'monitoring':='call'}
//Unique object ID
PROPERTY OID : OTCID
GET
END_GET
END_PROPERTY

{attribute 'monitoring':='call'}
PROPERTY PlanarMover : REFERENCE TO MC_PlanarMover
GET
END_GET
END_PROPERTY

{attribute 'monitoring':='call'}
PROPERTY PUBLIC ProductData : I_XP_ProductData
GET
END_GET
SET
END_SET
END_PROPERTY

END_INTERFACE

// COMPONENTs/Track/I_XP_Track
INTERFACE I_XP_Track  EXTENDS __SYSTEM.IQueryInterface, I_CH_Object

METHOD AddMover : HRESULT
VAR_INPUT
	ipMover : I_XP_Mover;
END_VAR
END_METHOD

METHOD AddToGroup : HRESULT
VAR_INPUT
	iGroup : I_XP_Group;
END_VAR
END_METHOD

{attribute 'monitoring':='call'}
PROPERTY ClosedLoop : BOOL
GET
END_GET
END_PROPERTY

METHOD Configure : HRESULT
VAR_INPUT
END_VAR
END_METHOD

METHOD Configuring : HRESULT
VAR_INPUT
END_VAR
END_METHOD

{attribute 'monitoring':='call'}
PROPERTY CtsMoversOnTrack : UINT
GET
END_GET
END_PROPERTY

METHOD Disable : HRESULT
VAR_INPUT
END_VAR
END_METHOD

METHOD Enable : HRESULT
VAR_INPUT
END_VAR
END_METHOD

{attribute 'monitoring':='call'}
PROPERTY Feedback : I_XP_Feedback
GET
END_GET
END_PROPERTY

{attribute 'monitoring':='call'}
//[mm]
PROPERTY Length : LREAL
GET
END_GET
END_PROPERTY

{attribute 'monitoring':='call'}
//Unique object ID
PROPERTY OID : OTCID
GET
END_GET
END_PROPERTY

{attribute 'monitoring':='call'}
PROPERTY PlanarTrack : REFERENCE TO MC_PlanarTrack
GET
END_GET
END_PROPERTY

METHOD RemoveFromGroup : HRESULT
END_METHOD

METHOD Reset : HRESULT
VAR_INPUT
END_VAR
END_METHOD

{attribute 'monitoring':='call'}
//List of interfaces to stations on this track
PROPERTY StationsOnTrack : I_CH_List
GET
END_GET
END_PROPERTY

{attribute 'monitoring':='call'}
//List of interfaces from other tracks
PROPERTY TracksAhead : I_CH_List
GET
END_GET
END_PROPERTY

{attribute 'monitoring':='call'}
//List of interfaces from other tracks
PROPERTY TracksBehinde : I_CH_List
GET
END_GET
END_PROPERTY

{attribute 'monitoring':='call'}
PROPERTY TracksEndAtThis : REFERENCE TO  ARRAY[0..(XPlanarParameterlist.N_MAX_STATIONS_AHEAD_OR_BEHIND-1)] OF I_XP_Track
GET
END_GET
END_PROPERTY

{attribute 'monitoring':='call'}
PROPERTY TracksStartFromThis : REFERENCE TO ARRAY[0..(XPlanarParameterlist.N_MAX_STATIONS_AHEAD_OR_BEHIND-1)] OF I_XP_Track
GET
END_GET
END_PROPERTY

END_INTERFACE

// COMPONENTs/Mover/I_XP_Mover
INTERFACE I_XP_Mover  EXTENDS __SYSTEM.IQueryInterface, I_CH_Object

METHOD AddToGroup : HRESULT
VAR_INPUT
	iGroup : I_XP_Group;
END_VAR
END_METHOD

METHOD RemoveFromGroup : HRESULT
END_METHOD

METHOD Halt : HRESULT
VAR_INPUT
END_VAR
END_METHOD

METHOD MoveA : HRESULT
VAR_INPUT
	fPosition : LREAL;
END_VAR
END_METHOD

METHOD MoveB : HRESULT
VAR_INPUT
	fPosition : LREAL;
END_VAR
END_METHOD

METHOD MoveC : HRESULT
VAR_INPUT
	fPosition : LREAL;
	
	(* Addition turns to move in modulo movement (positive or negative). *)
	additionalTurns : UDINT := 0;
	
	(* Direction in which the target is approached. *)
	direction : Tc3_Mc3Definitions.MC_DIRECTION := Tc3_Mc3Definitions.MC_DIRECTION.mcDirectionNonModulo;
END_VAR
END_METHOD

METHOD MoveXY : HRESULT
VAR_INPUT
	fPosition_X : LREAL;
	fPosition_Y : LREAL;
END_VAR
END_METHOD

METHOD MoveZ : HRESULT
VAR_INPUT
	fPosition : LREAL;
END_VAR
END_METHOD

METHOD Disable : HRESULT
VAR_INPUT
END_VAR
END_METHOD

METHOD Enable : HRESULT
VAR_INPUT
END_VAR
END_METHOD

METHOD Reset : HRESULT
VAR_INPUT
END_VAR
END_METHOD

{attribute 'monitoring':='call'}
PROPERTY CurrentTrack : I_XP_Track
GET
END_GET
END_PROPERTY

METHOD DistToTrack : LREAL
VAR_INPUT
	iTrack : I_XP_Track;
END_VAR
END_METHOD

METHOD JoinTrack : HRESULT
VAR_INPUT
	iTrack : I_XP_Track;
END_VAR
END_METHOD

{attribute 'monitoring':='call'}
PROPERTY LastCmdTargedGap : LREAL
GET
END_GET
END_PROPERTY

{attribute 'monitoring':='call'}
PROPERTY LastCmdTargedPosition : LREAL
GET
END_GET
END_PROPERTY

{attribute 'monitoring':='call'}
PROPERTY LastCmdTargedTrack: I_XP_Track
GET
END_GET
END_PROPERTY

METHOD MoveOnTrack : HRESULT
VAR_INPUT
	ipTrack : I_XP_Track;
	fPosition : LREAL;
	fGap : LREAL;
END_VAR
END_METHOD

METHOD MoveOnTrack_ShortestWay : HRESULT
VAR_INPUT
	ipTrack : I_XP_Track;
	fPosition : LREAL;
	fGap : LREAL;
END_VAR
END_METHOD

METHOD MoveOnTrackToStation : HRESULT
VAR_INPUT
	ipStation : I_XP_Station;
	fGap : LREAL;
END_VAR
END_METHOD

{attribute 'monitoring':='call'}
PROPERTY ParentStation : I_XP_Station
GET
END_GET
SET
END_SET
END_PROPERTY

{attribute 'monitoring':='call'}
PROPERTY PositionOnTrack : Lreal
GET
END_GET
END_PROPERTY

{attribute 'monitoring':='call'}
PROPERTY TargetStation : String
GET
END_GET
SET
END_SET
END_PROPERTY

PROPERTY TcIoXPlanarMover : Tc3_XPlanarUtility.I_TcIoXPlanarMover
GET
END_GET
END_PROPERTY

{attribute 'monitoring':='call'}
PROPERTY UtilityMover : Tc3_XPlanarUtility.I_McPlanarMover
GET
END_GET
END_PROPERTY

{attribute 'monitoring':='call'}
PROPERTY DistToParentStation : LREAL //Distance to the responsible parent station [mm]
GET
END_GET
END_PROPERTY

{attribute 'OPC.UA.DA.Property' := '1'}
{attribute 'monitoring':='call'}
PROPERTY Feedback : I_XP_Feedback
GET
END_GET
END_PROPERTY

{attribute 'monitoring':='call'}
PROPERTY Mapped : BOOL //Project is mapped to MC (McToPlc and PlcToMc)
GET
END_GET
END_PROPERTY

{attribute 'monitoring':='call'}
PROPERTY Mode : MC_PLANAR_MOVER_COMMAND_MODE
GET
END_GET
END_PROPERTY

{attribute 'monitoring':='call'}
//Unique object ID
PROPERTY OID : OTCID
GET
END_GET
END_PROPERTY

{attribute 'monitoring':='call'}
PROPERTY PlanarMover : REFERENCE TO MC_PlanarMover
GET
END_GET
END_PROPERTY

{attribute 'monitoring':='call'}
PROPERTY Route : REFERENCE TO FB_CH_List
GET
END_GET
END_PROPERTY

END_INTERFACE

// COMPONENTs/Stationen/I_XP_Station
INTERFACE I_XP_Station EXTENDS __SYSTEM.IQueryInterface, I_CH_Object

{attribute 'monitoring':='call'}
//Track on which the station is located
PROPERTY AccocietedTrack : I_XP_Track
GET
END_GET
END_PROPERTY

METHOD AddMoverToQueue : HRESULT
VAR_INPUT
	ipMover : I_XP_Mover;
END_VAR
END_METHOD

{attribute 'monitoring':='call'}
//List of movers managed by this station
PROPERTY AssignedMovers : I_CH_List
GET
END_GET
END_PROPERTY

//Call this Methode whith seq 0->100, and wait each step until S_OK is returned
METHOD Configure : HRESULT
VAR_INPUT
	nSeq : UINT; //0->100
END_VAR
END_METHOD

{attribute 'monitoring':='call'}
PROPERTY CtsEmptySpaceInQueue : UDINT
GET
END_GET
END_PROPERTY

METHOD DeleteMoversQueue : HRESULT
VAR_INPUT
END_VAR
END_METHOD

{attribute 'monitoring':='call'}
PROPERTY Filter : STRING
GET
END_GET
SET
END_SET
END_PROPERTY

{attribute 'monitoring':='call'}
//List of paths that lead to stations before this station
PROPERTY PathsAhead : I_CH_List
GET
END_GET
END_PROPERTY

{attribute 'monitoring':='call'}
//List of paths that lead to stations behind this station
PROPERTY PathsBehinde : I_CH_List
GET
END_GET
END_PROPERTY

{attribute 'monitoring':='call'}
//[mm] from the beginning of the assigned track
PROPERTY PositionOnTrack : LREAL
GET
END_GET
END_PROPERTY

{attribute 'monitoring':='call'}
//Position on the assigned track
PROPERTY PositionOnTrackXY : REFERENCE TO PositionXY
GET
END_GET
END_PROPERTY

{attribute 'monitoring':='call'}
//Planned position, not necessarily on the track
PROPERTY PositionXY : REFERENCE TO  PositionXY
GET
END_GET
END_PROPERTY

{attribute 'monitoring':='call'}
//prevent further movers from entering the station, 
//e.g. to prevent a collision. All movers that are already moving to reach this station will be stopped with a stop 
//and restarted with Ready True.
PROPERTY ReadyToRecvMovers : BOOL
GET
END_GET
END_PROPERTY

METHOD SearchNextBestStationByName : ST_PathFinder_1
VAR_INPUT
	sTargedStation : STRING; //unique station name or group of stations
	nPermittedSearchDepth : UINT;
	bCallFromExternal: BOOL; //set to true for an external call. set to false for a recursive call
END_VAR
END_METHOD

METHOD SendMoversToStation : I_CH_Feedback //All movers in the station are sent to this destination
VAR_INPUT
	sTargetStation: STRING;//unique station name or group of stations
END_VAR
END_METHOD

{attribute 'monitoring':='call'}
//List of stations before this station
PROPERTY StationsAhead : I_CH_List
GET
END_GET
END_PROPERTY

{attribute 'monitoring':='call'}
//List of stations behinde this station
PROPERTY StationsBehinde : I_CH_List
GET
END_GET
END_PROPERTY

{attribute 'monitoring':='call'}
PROPERTY TargetGroupe : STRING
GET
END_GET
END_PROPERTY

METHOD Update : HRESULT
VAR_INPUT
END_VAR
END_METHOD

END_INTERFACE

// COMPONENTs/Mover/FB_XP_Mover
// The warning " Interface of overridden methode xxx of base I_xxx doesn't match declaration" can be disabled here. 
{warning disable C0094 }
{attribute 'no_explicit_call' := 'Do not call the body - Stick to OOP'}
(* XPlanar mover - n per associated XPlanar. Can be instantiated as an array and/or individually
	The Planar mover is a software object that represents an XPlanar mover. It summarizes the state of the real mover (position, velocity, etc.) 
	for the user. In addition, the user has the possibility to influence or control the state of the real mover via the Planar mover. *)	
FUNCTION_BLOCK FB_XP_Mover EXTENDS FB_CH_Object IMPLEMENTS I_XP_Mover, I_XP_Mover_PLC
VAR
	fbRoute : FB_CH_List;
END_VAR

VAR
	//Link to MC-Mover
	fbMover : MC_PlanarMover;
	
	{attribute 'hide'}  
	bInitDone :BOOL := FALSE;
	{attribute 'hide'}               	
	fbFeedback 			: FB_XP_Feedback;
	{attribute 'hide'}                   	
	eActiveCommand 		: CHALET_Nc.E_NcAxisCommands := CHALET_Nc.E_NcAxisCommands.None;
	{attribute 'hide'} 
	fbUtilityMover : FB_McPlanarMover;
	{attribute 'hide'}
	iXpSystem : I_XP_System_Registration;
	{attribute 'hide'} 
	sTargedStation : STRING;
	{attribute 'hide'} 
	sCurrentStation : STRING;
	{attribute 'hide'}
	ipParentStation : I_XP_Station; //This is the station in which the Mover is currently standing or moving.	
	{attribute 'hide'}
	fLastCmdTargedPosition : LREAL; //the last commanded target position [mm]
	{attribute 'hide'}	
	fLastCmdTargedGap 	: LREAL; //the last commanded target gap
	{attribute 'hide'}		
//	fDistToParentStation : LREAL; //Distance to the responsible parent station [mm]
	{attribute 'hide'}		
	ipLastCmdTrack : I_XP_Track;
	{attribute 'hide'}
	ipProductData : I_XP_ProductData; //later the required interface of the tool or product can be queried via query interface
END_VAR

//External Setpoint Generator
VAR
	AxisSetpointX : FB_NcAxis;
	AxisSetpointY : FB_NcAxis;
	AxisSetpointZ : FB_NcAxis;
	AxisSetpointA : FB_NcAxis;
	AxisSetpointB : FB_NcAxis;
	AxisSetpointC : FB_NcAxis;
END_VAR


//DynamicConstraint
VAR
	{attribute 'hide'} 
	fbDynConstraintContainer 	: DynamicConstraint_Container;		//A container for dynamic constraints.
	{attribute 'hide'} 
	fbDynConstraintPath 		: DynamicConstraint_PathXY; 		//One dimensional dynamic constraint along the XY-components of a path, ignoring non-tangential effects.
	{attribute 'hide'} 	
	fbDynConstraintCoordinates	: DynamicConstraint_Coordinates;	//Dynamic constraints for individual coordinates.
END_VAR


// Planar-Feedback objects
VAR
	{attribute 'hide'} 
	fbFeedbackMoveA : MC_PlanarFeedback;
	{attribute 'hide'} 
	fbFeedbackMoveB : MC_PlanarFeedback;
	{attribute 'hide'} 
	fbFeedbackMoveC : MC_PlanarFeedback;
	{attribute 'hide'} 
	fbFeedbackMoveXY : MC_PlanarFeedback;
	{attribute 'hide'} 
	fbFeedbackMoveZ : MC_PlanarFeedback;
	{attribute 'hide'} 
	fbFeedbackEnable : MC_PlanarFeedback;
	{attribute 'hide'} 
	fbFeedbackDisable : MC_PlanarFeedback;
	{attribute 'hide'} 
	fbFeedbackHalt : MC_PlanarFeedback;
	{attribute 'hide'} 
	fbFeedbackReset : MC_PlanarFeedback;
	{attribute 'hide'} 
	fbFeedbackAddToGrp : MC_PlanarFeedback;
	{attribute 'hide'} 
	fbFeedbackRmvFromGrp : MC_PlanarFeedback;
	{attribute 'hide'} 
	fbFeedbackJoinTrack : MC_PlanarFeedback;
	{attribute 'hide'} 
	fbFeedbackMoveOnTrack: MC_PlanarFeedback;	
	{attribute 'hide'} 
	fbFeedbackExtStart : MC_PlanarFeedback;
	{attribute 'hide'} 
	fbFeedbackExtStop : MC_PlanarFeedback;
END_VAR
{warning restore C0094}

PROPERTY DynConstraint : REFERENCE TO DynamicConstraint_Container
GET
DynConstraint REF= THIS^.fbDynConstraintContainer;
END_GET
END_PROPERTY

METHOD SetDynConstraint_A : BOOL //Dynamic constraints for individual coordinates.
VAR_INPUT
    V : MC_LREAL; //equivalent to data type LREAL + MC_DEFAULT, MC_MAXIMUM
    A : MC_LREAL; //equivalent to data type LREAL + MC_DEFAULT, MC_MAXIMUM
    D : MC_LREAL; //equivalent to data type LREAL + MC_DEFAULT, MC_MAXIMUM
    J : MC_LREAL; //equivalent to data type LREAL + MC_DEFAULT, MC_MAXIMUM
END_VAR
THIS^.fbDynConstraintCoordinates.SetLimit(	Coordinate := Coord_Mcs_A1, 
											V := V, 
											A := A, 
											D := D, 
											J := J);
											
//Changes to the origin constraint do not affect the copy of the constraint in the instance of the DynamicConstraint_Container.
//For this reason, the container is being refreshed here							
fbDynConstraintContainer.Clear();
fbDynConstraintContainer.AddConstraint(fbDynConstraintPath);
fbDynConstraintContainer.AddConstraint(fbDynConstraintCoordinates);
END_METHOD

METHOD SetDynConstraint_B : BOOL //Dynamic constraints for individual coordinates.
VAR_INPUT
    V : MC_LREAL; //equivalent to data type LREAL + MC_DEFAULT, MC_MAXIMUM
    A : MC_LREAL; //equivalent to data type LREAL + MC_DEFAULT, MC_MAXIMUM
    D : MC_LREAL; //equivalent to data type LREAL + MC_DEFAULT, MC_MAXIMUM
    J : MC_LREAL; //equivalent to data type LREAL + MC_DEFAULT, MC_MAXIMUM
END_VAR
THIS^.fbDynConstraintCoordinates.SetLimit(	Coordinate := Coord_Mcs_B1, 
											V := V, 
											A := A, 
											D := D, 
											J := J);											

//Changes to the origin constraint do not affect the copy of the constraint in the instance of the DynamicConstraint_Container.
//For this reason, the container is being refreshed here							
fbDynConstraintContainer.Clear();
fbDynConstraintContainer.AddConstraint(fbDynConstraintPath);
fbDynConstraintContainer.AddConstraint(fbDynConstraintCoordinates);
END_METHOD

METHOD SetDynConstraint_C : BOOL //Dynamic constraints for individual coordinates.
VAR_INPUT
    V : MC_LREAL; //equivalent to data type LREAL + MC_DEFAULT, MC_MAXIMUM
    A : MC_LREAL; //equivalent to data type LREAL + MC_DEFAULT, MC_MAXIMUM
    D : MC_LREAL; //equivalent to data type LREAL + MC_DEFAULT, MC_MAXIMUM
    J : MC_LREAL; //equivalent to data type LREAL + MC_DEFAULT, MC_MAXIMUM
END_VAR
THIS^.fbDynConstraintCoordinates.SetLimit(	Coordinate := Coord_Mcs_C1, 
											V := V, 
											A := A, 
											D := D, 
											J := J);											

//Changes to the origin constraint do not affect the copy of the constraint in the instance of the DynamicConstraint_Container.
//For this reason, the container is being refreshed here							
fbDynConstraintContainer.Clear();
fbDynConstraintContainer.AddConstraint(fbDynConstraintPath);
fbDynConstraintContainer.AddConstraint(fbDynConstraintCoordinates);
END_METHOD

METHOD SetDynConstraint_Path : BOOL //One dimensional dynamic constraint along the XY-components of a path, ignoring non-tangential effects.
VAR_INPUT
    V : MC_LREAL; //equivalent to data type LREAL + MC_DEFAULT, MC_MAXIMUM
    A : MC_LREAL; //equivalent to data type LREAL + MC_DEFAULT, MC_MAXIMUM
    D : MC_LREAL; //equivalent to data type LREAL + MC_DEFAULT, MC_MAXIMUM
    J : MC_LREAL; //equivalent to data type LREAL + MC_DEFAULT, MC_MAXIMUM
END_VAR
THIS^.fbDynConstraintPath.SetValuesVADJ(V := V, 
										A := A, 
										D := D, 
										J := J);											

//Changes to the origin constraint do not affect the copy of the constraint in the instance of the DynamicConstraint_Container.
//For this reason, the container is being refreshed here							
fbDynConstraintContainer.Clear();
fbDynConstraintContainer.AddConstraint(fbDynConstraintPath);
fbDynConstraintContainer.AddConstraint(fbDynConstraintCoordinates);
END_METHOD

METHOD SetDynConstraint_X : BOOL //Dynamic constraints for individual coordinates.
VAR_INPUT
    V : MC_LREAL; //equivalent to data type LREAL + MC_DEFAULT, MC_MAXIMUM
    A : MC_LREAL; //equivalent to data type LREAL + MC_DEFAULT, MC_MAXIMUM
    D : MC_LREAL; //equivalent to data type LREAL + MC_DEFAULT, MC_MAXIMUM
    J : MC_LREAL; //equivalent to data type LREAL + MC_DEFAULT, MC_MAXIMUM
END_VAR
THIS^.fbDynConstraintCoordinates.SetLimit(	Coordinate := Coord_Mcs_X, 
											V := V, 
											A := A, 
											D := D, 
											J := J);											

//Changes to the origin constraint do not affect the copy of the constraint in the instance of the DynamicConstraint_Container.
//For this reason, the container is being refreshed here							
fbDynConstraintContainer.Clear();
fbDynConstraintContainer.AddConstraint(fbDynConstraintPath);
fbDynConstraintContainer.AddConstraint(fbDynConstraintCoordinates);
END_METHOD

METHOD SetDynConstraint_Y : BOOL //Dynamic constraints for individual coordinates.
VAR_INPUT
    V : MC_LREAL; //equivalent to data type LREAL + MC_DEFAULT, MC_MAXIMUM
    A : MC_LREAL; //equivalent to data type LREAL + MC_DEFAULT, MC_MAXIMUM
    D : MC_LREAL; //equivalent to data type LREAL + MC_DEFAULT, MC_MAXIMUM
    J : MC_LREAL; //equivalent to data type LREAL + MC_DEFAULT, MC_MAXIMUM
END_VAR
THIS^.fbDynConstraintCoordinates.SetLimit(	Coordinate := Coord_Mcs_Y, 
											V := V, 
											A := A, 
											D := D, 
											J := J);											

//Changes to the origin constraint do not affect the copy of the constraint in the instance of the DynamicConstraint_Container.
//For this reason, the container is being refreshed here							
fbDynConstraintContainer.Clear();
fbDynConstraintContainer.AddConstraint(fbDynConstraintPath);
fbDynConstraintContainer.AddConstraint(fbDynConstraintCoordinates);
END_METHOD

METHOD SetDynConstraint_Z : BOOL //Dynamic constraints for individual coordinates.
VAR_INPUT
    V : MC_LREAL; //equivalent to data type LREAL + MC_DEFAULT, MC_MAXIMUM
    A : MC_LREAL; //equivalent to data type LREAL + MC_DEFAULT, MC_MAXIMUM
    D : MC_LREAL; //equivalent to data type LREAL + MC_DEFAULT, MC_MAXIMUM
    J : MC_LREAL; //equivalent to data type LREAL + MC_DEFAULT, MC_MAXIMUM
END_VAR
THIS^.fbDynConstraintCoordinates.SetLimit(	Coordinate := Coord_Mcs_Z, 
											V := MC_DEFAULT, 
											A := A, 
											D := D, 
											J := J);											

//Changes to the origin constraint do not affect the copy of the constraint in the instance of the DynamicConstraint_Container.
//For this reason, the container is being refreshed here							
fbDynConstraintContainer.Clear();
fbDynConstraintContainer.AddConstraint(fbDynConstraintPath);
fbDynConstraintContainer.AddConstraint(fbDynConstraintCoordinates);
END_METHOD

{attribute 'monitoring':='call'}
PROPERTY  AxisExtSetpointA : CHALET_Nc.I_NcAxis_PLC
GET
AxisExtSetpointA := THIS^.AxisSetpointA;
END_GET
END_PROPERTY

{attribute 'monitoring':='call'}
PROPERTY AxisExtSetpointB : CHALET_Nc.I_NcAxis_PLC
GET
AxisExtSetpointB := THIS^.AxisSetpointB;
END_GET
END_PROPERTY

{attribute 'monitoring':='call'}
PROPERTY AxisExtSetpointC : CHALET_Nc.I_NcAxis_PLC
GET
AxisExtSetpointC := THIS^.AxisSetpointC;
END_GET
END_PROPERTY

{attribute 'monitoring':='call'}
PROPERTY  AxisExtSetpointX : CHALET_Nc.I_NcAxis_PLC
GET
AxisExtSetpointX := THIS^.AxisSetpointX;
END_GET
END_PROPERTY

{attribute 'monitoring':='call'}
PROPERTY AxisExtSetpointY : CHALET_Nc.I_NcAxis_PLC
GET
AxisExtSetpointY := THIS^.AxisSetpointY;
END_GET
END_PROPERTY

{attribute 'monitoring':='call'}
PROPERTY AxisExtSetpointZ : CHALET_Nc.I_NcAxis_PLC
GET
AxisExtSetpointZ := THIS^.AxisSetpointZ;
END_GET
END_PROPERTY

METHOD StartExternalSetpoint : HRESULT
VAR
	startOptions : ST_ExternalSetpointGenerationOptions;
END_VAR
IF THIS^.fbMover.Error THEN
	THIS^.fbFeedback.LastCommandAccepted	:= FALSE;
	//Error active/not ready

// Check, that all axis standing on 0.0
ELSIF (AxisSetpointX.SetPosition <> 0.0 OR AxisSetpointY.SetPosition <> 0.0  OR AxisSetpointZ.SetPosition <> 0.0  OR AxisSetpointA.SetPosition <> 0.0  OR AxisSetpointB.SetPosition <> 0.0  OR AxisSetpointC.SetPosition <> 0.0) THEN
	THIS^.fbFeedback.LastCommandAccepted	:= FALSE;
	//Error, to prevent the mover from making a jump in relative mode, each axis should be set to position 0 		
	
ELSIF (AxisSetpointX.Mapped AND AxisSetpointX.Feedback.Error) OR
		(AxisSetpointY.Mapped AND AxisSetpointY.Feedback.Error) OR
		(AxisSetpointZ.Mapped AND AxisSetpointZ.Feedback.Error) OR
		(AxisSetpointA.Mapped AND AxisSetpointA.Feedback.Error) OR
		(AxisSetpointB.Mapped AND AxisSetpointB.Feedback.Error) OR
		(AxisSetpointC.Mapped AND AxisSetpointC.Feedback.Error) THEN
	THIS^.fbFeedback.LastCommandAccepted	:= FALSE;
	//Axis Error active
	
ELSE

	THIS^.eActiveCommand 				:= CHALET_NC.E_NcAxisCommands.StartExternalSetpoint;
	THIS^.fbFeedback.LastCommandAccepted:= TRUE;		
	THIS^.fbFeedback.Busy 				:= TRUE;
	
	AxisSetpointX.PowerOn();
	AxisSetpointY.PowerOn();
	AxisSetpointZ.PowerOn();
	AxisSetpointA.PowerOn();
	AxisSetpointB.PowerOn();
	AxisSetpointC.PowerOn();

	startOptions.mode := MC_EXTERNAL_SET_POSITION_MODE.Relative;
	THIS^.fbMover.StartExternalSetpointGeneration(THIS^.fbFeedbackExtStart,startOptions);
	
	StartExternalSetpoint := S_OK;	
END_IF
END_METHOD

METHOD StopExternalSetpoint : HRESULT
VAR_INPUT
END_VAR
AxisSetpointX.PowerOff();
AxisSetpointY.PowerOff();
AxisSetpointZ.PowerOff();
AxisSetpointA.PowerOff();
AxisSetpointB.PowerOff();
AxisSetpointC.PowerOff();


THIS^.eActiveCommand 				:= CHALET_NC.E_NcAxisCommands.StopExternalSetpoint;
THIS^.fbFeedback.LastCommandAccepted:= TRUE;		
THIS^.fbFeedback.Busy 				:= TRUE;

THIS^.fbMover.StopExternalSetpointGeneration(THIS^.fbFeedbackExtStop);
StopExternalSetpoint := S_OK;
END_METHOD

METHOD PROTECTED UpdateExternalSetpoint : HRESULT
VAR_INPUT
END_VAR
VAR
	SetPos, SetVelo, SetAcc : MoverVector;
END_VAR
SetPos.X := AxisSetpointX.SetPosition;
SetPos.Y := AxisSetpointY.SetPosition;
SetPos.Z := AxisSetpointZ.SetPosition;
SetPos.A := AxisSetpointA.SetPosition;
SetPos.B := AxisSetpointB.SetPosition;
SetPos.C := AxisSetpointC.SetPosition;

SetVelo.X := AxisSetpointX.SetVelocity;
SetVelo.Y := AxisSetpointY.SetVelocity;
SetVelo.Z := AxisSetpointZ.SetVelocity;
SetVelo.A := AxisSetpointA.SetVelocity;
SetVelo.B := AxisSetpointB.SetVelocity;
SetVelo.C := AxisSetpointC.SetVelocity;

SetAcc.X := AxisSetpointX.Setacceleration;
SetAcc.Y := AxisSetpointY.Setacceleration;
SetAcc.Z := AxisSetpointZ.Setacceleration;
SetAcc.A := AxisSetpointA.Setacceleration;
SetAcc.B := AxisSetpointB.Setacceleration;
SetAcc.C := AxisSetpointC.Setacceleration;

IF THIS^.fbMover.MCTOPLC.STD.State = MC_PLANAR_STATE.Enabled THEN
	THIS^.fbMover.SetExternalSetpoint(	setPosition 		:= SetPos, 
										setVelocity 		:= SetVelo,
										setAcceleration 	:= SetAcc);
END_IF



IF AxisSetpointX.Mapped THEN AxisSetpointX.Update() ;END_IF
IF AxisSetpointY.Mapped THEN AxisSetpointY.Update() ;END_IF
IF AxisSetpointZ.Mapped THEN AxisSetpointZ.Update() ;END_IF
IF AxisSetpointA.Mapped THEN AxisSetpointA.Update() ;END_IF
IF AxisSetpointB.Mapped THEN AxisSetpointB.Update() ;END_IF
IF AxisSetpointC.Mapped THEN AxisSetpointC.Update() ;END_IF
END_METHOD

METHOD AddToGroup : HRESULT
VAR_INPUT
	iGroup : I_XP_Group;
END_VAR
IF NOT THIS^.fbFeedback.Busy THEN
	THIS^.eActiveCommand 				:= CHALET_NC.E_NcAxisCommands.AddToGroupe;
	THIS^.fbFeedback.LastCommandAccepted:= TRUE;		
	THIS^.fbFeedback.Busy 				:= TRUE;
	
	iGroup.AddMover(THIS^.fbMover, THIS^.fbFeedbackAddToGrp);
	AddToGroup := S_OK;
ELSE
	AddToGroup := S_FALSE;
	THIS^.fbFeedback.LastCommandAccepted:= FALSE;	
END_IF
END_METHOD

METHOD RemoveFromGroup : HRESULT

VAR
	iGroup: INT;
END_VAR
IF NOT THIS^.fbFeedback.Busy THEN
	THIS^.eActiveCommand 				:= CHALET_NC.E_NcAxisCommands.RemoveFromGroupe;
	THIS^.fbFeedback.LastCommandAccepted:= TRUE;		
	THIS^.fbFeedback.Busy 				:= TRUE;
	
	THIS^.fbMover.RemoveFromGroup(THIS^.fbFeedbackRmvFromGrp);
	
	RemoveFromGroup := S_OK;
ELSE
	RemoveFromGroup := S_FALSE;
	THIS^.fbFeedback.LastCommandAccepted:= FALSE;	
END_IF
END_METHOD

METHOD Halt : HRESULT
VAR_INPUT
END_VAR
THIS^.eActiveCommand 				:= CHALET_NC.E_NcAxisCommands.Halt;
THIS^.fbFeedback.LastCommandAccepted:= TRUE;		
THIS^.fbFeedback.Busy 				:= TRUE;

THIS^.fbMover.Halt(	commandFeedback := THIS^.fbFeedbackHalt, 
					constraint 		:= THIS^.fbDynConstraintContainer 
				   );

Halt := S_OK;
END_METHOD

METHOD MoveA : HRESULT
VAR_INPUT
	fPosition : LREAL;
END_VAR
THIS^.eActiveCommand 				:= CHALET_NC.E_NcAxisCommands.MoveA;
THIS^.fbFeedback.LastCommandAccepted:= TRUE;		
THIS^.fbFeedback.Busy 				:= TRUE;

THIS^.fbMover.MoveA(commandFeedback	:= THIS^.fbFeedbackMoveA, 
					targetPosition	:= fPosition, 
					constraint		:= THIS^.fbDynConstraintContainer
					);

MoveA := S_OK;
END_METHOD

METHOD MoveB : HRESULT
VAR_INPUT
	fPosition : LREAL;
END_VAR
THIS^.eActiveCommand 				:= CHALET_NC.E_NcAxisCommands.MoveB;
THIS^.fbFeedback.LastCommandAccepted:= TRUE;		
THIS^.fbFeedback.Busy 				:= TRUE;

THIS^.fbMover.MoveB(commandFeedback	:= THIS^.fbFeedbackMoveB, 
					targetPosition	:= fPosition, 
					constraint		:= THIS^.fbDynConstraintContainer
					);

MoveB := S_OK;
END_METHOD

METHOD MoveC : HRESULT
VAR_INPUT
	fPosition : LREAL;
	
	(* Addition turns to move in modulo movement (positive or negative). *)
	additionalTurns : UDINT := 0;
	
	(* Direction in which the target is approached. *)
	direction : Tc3_Mc3Definitions.MC_DIRECTION := Tc3_Mc3Definitions.MC_DIRECTION.mcDirectionNonModulo;
END_VAR
VAR
	stMoveCOptions : ST_MoveCOptions;
END_VAR
THIS^.eActiveCommand 				:= CHALET_NC.E_NcAxisCommands.MoveC;
THIS^.fbFeedback.LastCommandAccepted:= TRUE;		
THIS^.fbFeedback.Busy 				:= TRUE;


stMoveCOptions.additionalTurns := additionalTurns;
stMoveCOptions.direction := direction;


THIS^.fbMover.MoveC(commandFeedback	:= THIS^.fbFeedbackMoveC, 
					targetPosition	:= fPosition, 
					constraint		:= THIS^.fbDynConstraintContainer, 
					options			:= stMoveCOptions
					);

MoveC := S_OK;
END_METHOD

METHOD MoveXY : HRESULT
VAR_INPUT
	fPosition_X : LREAL;
	fPosition_Y : LREAL;
END_VAR
VAR
	fbTargetPosition 	: PositionXYC;
	stMoveOptions 		: ST_MoveToPositionOptions;
END_VAR
THIS^.eActiveCommand 				:= CHALET_NC.E_NcAxisCommands.MoveXY;
THIS^.fbFeedback.LastCommandAccepted:= TRUE;		
THIS^.fbFeedback.Busy 				:= TRUE;



fbTargetPosition.SetValuesXY(x := fPosition_X, y := fPosition_Y);

stMoveOptions.useOrientation := FALSE;

THIS^.fbMover.MoveToPosition(	commandFeedback	:= THIS^.fbFeedbackMoveXY, 
								targetPosition	:= fbTargetPosition,
								constraint		:= THIS^.fbDynConstraintContainer, 
								options			:= stMoveOptions);

MoveXY := S_OK;
END_METHOD

METHOD MoveZ : HRESULT
VAR_INPUT
	fPosition : LREAL;
END_VAR
THIS^.eActiveCommand 				:= CHALET_NC.E_NcAxisCommands.MoveZ;
THIS^.fbFeedback.LastCommandAccepted:= TRUE;		
THIS^.fbFeedback.Busy 				:= TRUE;


THIS^.fbMover.MoveZ(commandFeedback	:= THIS^.fbFeedbackMoveZ, 
					targetPosition	:= fPosition, 
					constraint		:= THIS^.fbDynConstraintContainer
					);

MoveZ := S_OK;
END_METHOD

METHOD Disable : HRESULT
VAR_INPUT
END_VAR
THIS^.eActiveCommand 				:= CHALET_NC.E_NcAxisCommands.Disable;
THIS^.fbFeedback.LastCommandAccepted:= TRUE;		
THIS^.fbFeedback.Busy 				:= TRUE;

THIS^.fbMover.Disable(THIS^.fbFeedbackDisable);
Disable := S_OK;
END_METHOD

METHOD Enable : HRESULT
VAR_INPUT
END_VAR
IF NOT THIS^.fbFeedback.Busy THEN
	THIS^.eActiveCommand 				:= CHALET_NC.E_NcAxisCommands.Enable;
	THIS^.fbFeedback.LastCommandAccepted:= TRUE;		
	THIS^.fbFeedback.Busy 				:= TRUE;

	THIS^.fbMover.Enable(fbFeedbackEnable);
	Enable := S_OK;
ELSE
	Enable := S_FALSE;
	THIS^.fbFeedback.LastCommandAccepted:= FALSE;	
END_IF
END_METHOD

METHOD Reset : HRESULT
VAR_INPUT
END_VAR
THIS^.eActiveCommand 				:= CHALET_NC.E_NcAxisCommands.Reset;
THIS^.fbFeedback.LastCommandAccepted:= TRUE;		
THIS^.fbFeedback.Busy 				:= TRUE;

THIS^.fbMover.Reset(THIS^.fbFeedbackReset);
Reset := S_OK;
END_METHOD

{attribute 'monitoring':='call'}
(* Indicates the command mode of an enabled PlanarMover, i.e. how setpoints are currently produced. *)
PROPERTY CommandMode : MC_PLANAR_MOVER_COMMAND_MODE
GET
CommandMode := THIS^.fbMover.MCTOPLC.STD.CommandMode;
END_GET
END_PROPERTY

{attribute 'monitoring':='call'}
(* Retruns lentgh of hypotenuse of the x and y error. (>=0[mm]) *)
PROPERTY LagDistanceXY : LREAL
GET
VAR
	fErrorX, fErrorY : LREAL;
END_VAR
// Set - Act
fErrorX := THIS^.fbMover.MCTOPLC.SET.SetPos.X - THIS^.fbMover.MCTOPLC.ACT.ActPos.X;
fErrorY := THIS^.fbMover.MCTOPLC.SET.SetPos.Y - THIS^.fbMover.MCTOPLC.ACT.ActPos.Y;


//Dist to center. Phytagoras -> c = sqrt( A^2 + B^2)
LagDistanceXY := SQRT(EXPT(fErrorX,2) + EXPT(fErrorY,2));
END_GET
END_PROPERTY

{attribute 'monitoring':='call'}
(* Contains the information of the Planar Mover passed from MC to PLC. XYZABC [mm] *)
PROPERTY PositionAct : REFERENCE TO MoverVector
GET
VAR_INST
	{attribute 'hide'}
	copyOfActPosition :  MoverVector;
END_VAR
//Creat an copy of the struct to view value in targeddbrowser and plc online view
copyOfActPosition := THIS^.fbMover.MCTOPLC.ACT.ActPos;
PositionAct REF= copyOfActPosition;
END_GET
END_PROPERTY

{attribute 'monitoring':='call'}
(* Provides the current planar mover setpoint XYZABC [mm] *)
PROPERTY PositionSet : REFERENCE TO MoverVector
GET
VAR_INST
	{attribute 'hide'}
	copyOfSetPosition :  MoverVector;
END_VAR
//Creat an copy of the struct to view value in targeddbrowser and plc online view
copyOfSetPosition := THIS^.fbMover.MCTOPLC.SET.SetPos;
PositionSet REF= copyOfSetPosition;
END_GET
END_PROPERTY

{attribute 'monitoring':='call'}
PROPERTY CurrentTrack : I_XP_Track
GET
VAR
	ipTrackObj : I_CH_Object;
	ipTrack : I_XP_Track;
END_VAR
IF iXpSystem <> 0 THEN
	ipTrackObj := iXpSystem.Tracks.FindOID(THIS^.PlanarMover.MCTOPLC.SETONTRACK.TrackOID);
	ToXpTrack(ipTrackObj,ipTrack);
END_IF

CurrentTrack := ipTrack;
END_GET
END_PROPERTY

METHOD DistToTrack : LREAL
VAR_INPUT
	iTrack : I_XP_Track;
END_VAR
VAR
	fPositionOnTrack : LREAL;
	trackPosition, moverPosition : PositionXYC;
END_VAR
moverPosition.x := PositionSet.x;
moverPosition.y := PositionSet.y;
moverPosition.c := PositionSet.c;

//Get Pos on track in mm
fPositionOnTrack := iTrack.PlanarTrack.GetArcLengthClosestTo(geometry:=moverPosition);

//Convert pos on track in XY
iTrack.PlanarTrack.GetPositionAt(arcLength := fPositionOnTrack, position:=trackPosition);

//Get distance to mover
DistToTrack := SQRT(EXPT((trackPosition.x - moverPosition.x),2)+EXPT((trackPosition.y - moverPosition.y),2));
END_METHOD

METHOD JoinTrack : HRESULT
VAR_INPUT
	iTrack : I_XP_Track;
END_VAR
VAR
	joinTrackOptions : ST_JoinTrackOptions;
END_VAR
IF iTrack <> 0 THEN
	THIS^.eActiveCommand 				:= CHALET_NC.E_NcAxisCommands.JoinTrack;
	THIS^.fbFeedback.LastCommandAccepted:= TRUE;		
	THIS^.fbFeedback.Busy 				:= TRUE;

	joinTrackOptions.useOrientation := TRUE;	
	THIS^.fbMover.JoinTrack(commandFeedback	:= THIS^.fbFeedbackJoinTrack, 
								targetTrack	:= iTrack.PlanarTrack, 
								constraint	:= THIS^.fbDynConstraintContainer,
								options		:= joinTrackOptions);								
	JoinTrack := S_OK;
ELSE
	JoinTrack := S_FALSE;
	THIS^.fbFeedback.LastCommandAccepted:= FALSE;	
END_IF
END_METHOD

{attribute 'monitoring':='call'}
PROPERTY LastCmdTargedGap : LREAL
GET
LastCmdTargedGap := fLastCmdTargedGap;
END_GET
END_PROPERTY

{attribute 'monitoring':='call'}
PROPERTY LastCmdTargedPosition : LREAL
GET
LastCmdTargedPosition := fLastCmdTargedPosition;
END_GET
END_PROPERTY

{attribute 'monitoring':='call'}
PROPERTY LastCmdTargedTrack: I_XP_Track
GET
LastCmdTargedTrack := ipLastCmdTrack;
END_GET
END_PROPERTY

METHOD MoveOnTrack : HRESULT
VAR_INPUT
	ipTrack : I_XP_Track;
	fPosition : LREAL;
	fGap : LREAL;
END_VAR

VAR
	moveOptions: ST_MoveOnTrackOptions;
	//fMoverDiagonal : LREAL;
END_VAR
moveOptions.direction := Tc3_Mc3Definitions.MC_DIRECTION.mcDirectionPositive;
moveOptions.additionalTurns := 0;

//Use fix gap if requested gap is to small
moveOptions.gap := MAX(fGap, XPlanarParameterlist.F_MOVER_MINIMUM_GAP_ON_TRACK);

IF ipTrack <> 0 THEN
	THIS^.eActiveCommand 				:= CHALET_NC.E_NcAxisCommands.MoveOnTrack;
	THIS^.fbFeedback.LastCommandAccepted:= TRUE;		
	THIS^.fbFeedback.Busy 				:= TRUE;

	THIS^.fbMover.MoveOnTrack(
		commandFeedback			:= THIS^.fbFeedbackMoveOnTrack,
		targetTrack				:= ipTrack.PlanarTrack, 
		targetPositionOnTrack	:= fPosition, 
		constraint				:= THIS^.fbDynConstraintPath, 
		options					:= moveOptions);
	
	//Store the values
	fLastCmdTargedPosition 	:= fPosition; //the last commanded target position [mm]
	fLastCmdTargedGap 		:= moveOptions.gap; //the last commanded target gap
	ipLastCmdTrack		 	:= ipTrack; //the last commanded target track	
	
	
	MoveOnTrack := S_OK;
ELSE
	MoveOnTrack := S_FALSE;
	THIS^.fbFeedback.LastCommandAccepted:= FALSE;	
END_IF
END_METHOD

METHOD MoveOnTrack_ShortestWay : HRESULT
VAR_INPUT
	ipTrack : I_XP_Track;
	fPosition : LREAL;
	fGap : LREAL;
END_VAR

VAR
	moveOptions: ST_MoveOnTrackOptions;
	//fMoverDiagonal : LREAL;
END_VAR
moveOptions.direction := Tc3_Mc3Definitions.MC_DIRECTION.mcDirectionShortestWay;
moveOptions.additionalTurns := 0;

//Use fix gap if requested gap is to small
moveOptions.gap := MAX(fGap, XPlanarParameterlist.F_MOVER_MINIMUM_GAP_ON_TRACK);


IF ipTrack <> 0 THEN
	THIS^.eActiveCommand 				:= CHALET_NC.E_NcAxisCommands.MoveOnTrack;
	THIS^.fbFeedback.LastCommandAccepted:= TRUE;		
	THIS^.fbFeedback.Busy 				:= TRUE;
	
	THIS^.fbMover.MoveOnTrack(
		commandFeedback			:= THIS^.fbFeedbackMoveOnTrack,
		targetTrack				:= ipTrack.PlanarTrack, 
		targetPositionOnTrack	:= fPosition, 
		constraint				:= THIS^.fbDynConstraintPath, 
		options					:= moveOptions);
				
	fLastCmdTargedPosition 	:= fPosition; //the last commanded target position [mm]
	fLastCmdTargedGap 		:= moveOptions.gap; //the last commanded target gap
	ipLastCmdTrack		 	:= ipTrack; //the last commanded target track	
		
	MoveOnTrack_ShortestWay := S_OK;
ELSE
	MoveOnTrack_ShortestWay := S_FALSE;
	THIS^.fbFeedback.LastCommandAccepted:= FALSE;	
END_IF
END_METHOD

METHOD MoveOnTrackToStation : HRESULT
VAR_INPUT
	ipStation : I_XP_Station;
	fGap : LREAL;

END_VAR
IF ipStation <> 0 AND_THEN ipStation.AccocietedTrack <> 0 THEN

	MoveOnTrackToStation := MoveOnTrack(ipTrack:= ipStation.AccocietedTrack, 
										fPosition:= ipStation.PositionOnTrack, 
										fGap:= fGap);
ELSE
	MoveOnTrackToStation := E_FAIL;
	THIS^.fbFeedback.LastCommandAccepted:= FALSE;	
END_IF
END_METHOD

{attribute 'monitoring':='call'}
PROPERTY ParentStation : I_XP_Station
GET
ParentStation := ipParentStation;
END_GET
SET
ipParentStation := ParentStation;
END_SET
END_PROPERTY

{attribute 'monitoring':='call'}
PROPERTY PositionOnTrack : LREAL
GET
PositionOnTrack := THIS^.fbMover.MCTOPLC.SETONTRACK.SetPos;
END_GET
END_PROPERTY

{attribute 'monitoring':='call'}
PROPERTY TargetStation : STRING
GET
TargetStation := THIS^.sTargedStation;
END_GET
SET
THIS^.sTargedStation := TargetStation;
END_SET
END_PROPERTY

{attribute 'monitoring':='call'}
PROPERTY TcIoXPlanarMover : Tc3_XPlanarUtility.I_TcIoXPlanarMover
GET
VAR
	nLoopIndex : UINT;
	ipPlanarMover : I_TcIoXPlanarMover;
END_VAR
FOR nLoopIndex := 1 TO UDINT_TO_UINT(Param_TcIoXPlanarEnvironment.MaxXPlanarMoversPerXpu) DO
	ipPlanarMover := iXpSystem.Enviroment.UtilityEnvirement.XpuTcIo(1).MoverTcIo(nLoopIndex);
	IF ipPlanarMover <> 0 AND_THEN ipPlanarMover.GetNcMoverOid() = OID THEN
		TcIoXPlanarMover := iXpSystem.enviroment.UtilityEnvirement.XpuTcIo(1).MoverTcIo(nLoopIndex);
		RETURN;
	END_IF
END_FOR
END_GET
END_PROPERTY

{attribute 'monitoring':='call'}
PROPERTY UtilityMover : Tc3_XPlanarUtility.I_McPlanarMover
GET
UtilityMover := THIS^.fbUtilityMover;
END_GET
END_PROPERTY

{attribute 'monitoring':='call'}
//Distance to the responsible parent station [mm]
PROPERTY DistToParentStation : LREAL
GET
VAR
	fDistToParentStationTemp : LREAL := CHALET_BaseComponents.GVL_Datatypes.cMaxLreal;
	ipPath : I_XP_Path;
END_VAR
//Get distance to targed station
//check each path behind the parentstation if the mover is on it
THIS^.ParentStation.PathsBehinde.ResetIterator();
WHILE THIS^.ParentStation.PathsBehinde.HasNextObject() DO
	IF __QUERYINTERFACE(THIS^.ParentStation.PathsBehinde.GetNextObject(), ipPath) THEN
		//get shortest distance
		fDistToParentStationTemp:= MIN(ipPath.DistanceToDestiantion(ipTrack:= THIS^.CurrentTrack, fPosOnTrack := THIS^.PositionOnTrack), fDistToParentStationTemp);
	END_IF
END_WHILE
THIS^.ParentStation.PathsBehinde.RestoreIterator();


DistToParentStation := fDistToParentStationTemp;
END_GET
END_PROPERTY

METHOD FB_init : BOOL
VAR_INPUT
	bInitRetains : BOOL; // if TRUE, the retain variables are initialized (warm start / cold start)
	bInCopyCode : BOOL;  // if TRUE, the instance afterwards gets moved into the copy code (online change)
	
	
	ipSystem : I_CH_Object;
END_VAR
VAR_INST
	{attribute 'hide'}
	bFBInitCalledOnce : BOOL; //Do the following code once during start up and not during onlinechange
END_VAR
//Do the following code once during start up and not during onlinechange
IF NOT bFBInitCalledOnce THEN 
	
	
	(* Register to the Xplanar System
	   1. Test if the interface exists
	   2. Test if the object implements a "System for Mover" interface 
	*)
	IF ipSystem <> 0 AND_THEN __QUERYINTERFACE(ipSystem,THIS^.iXpSystem) THEN
		THIS^.iXpSystem.RegisterMover(THIS^);
	END_IF

END_IF

bFBInitCalledOnce := TRUE;
END_METHOD

{attribute 'monitoring':='call'}
PROPERTY Feedback : I_XP_Feedback
GET
Feedback := THIS^.fbFeedback;
END_GET
END_PROPERTY

METHOD Initialize : HRESULT
VAR
	bWaitForAxisInit : BOOL;
	hrExtAxis : HRESULT;
	stVarInfo : __SYSTEM.VAR_INFO;
END_VAR

VAR_INST
	//This error cannot be reset. Requires a reset cold
	{attribute 'hide'}	
	fbInitError : FB_TcAlarm;
END_VAR
// Check if link to MC-Mover is mapped
IF NOT THIS^.Mapped THEN
	IF NOT fbInitError.bRaised THEN 
		//This error cannot be reset. Requires a reset cold
		fbInitError.CreateEx(stEventEntry:=TC_EVENTS.CHALET_XPlanar_Events.VariableLinkMissing, ipSourceInfo := THIS^.fbSourceInfo, bWithConfirmation := FALSE);
		stVarInfo := __VARINFO(fbMover);
		fbInitError.ipArguments.AddString(stVarInfo.Symbol);
		fbInitError.Raise(0);
	END_IF
	Initialize := E_FAIL;
	RETURN;
END_IF


	
IF NOT bInitDone THEN
	//Set all move dynamic constraint to the axis default value.
	THIS^.SetDynConstraint_X(MC_DEFAULT,MC_DEFAULT,MC_DEFAULT,MC_DEFAULT);
	THIS^.SetDynConstraint_Y(MC_DEFAULT,MC_DEFAULT,MC_DEFAULT,MC_DEFAULT);	
	THIS^.SetDynConstraint_Z(MC_DEFAULT,MC_DEFAULT,MC_DEFAULT,MC_DEFAULT);	
	THIS^.SetDynConstraint_A(MC_DEFAULT,MC_DEFAULT,MC_DEFAULT,MC_DEFAULT);	
	THIS^.SetDynConstraint_B(MC_DEFAULT,MC_DEFAULT,MC_DEFAULT,MC_DEFAULT);
	THIS^.SetDynConstraint_C(MC_DEFAULT,MC_DEFAULT,MC_DEFAULT,MC_DEFAULT);
	THIS^.SetDynConstraint_Path(MC_DEFAULT,MC_DEFAULT,MC_DEFAULT,MC_DEFAULT);

	//Call Init of Setpointaxis only, if mapped
	IF AxisSetpointX.Mapped THEN hrExtAxis := GetMostSignificant(hrExtAxis, AxisSetpointX.Initialize());END_IF
	IF AxisSetpointY.Mapped THEN hrExtAxis := GetMostSignificant(hrExtAxis, AxisSetpointY.Initialize());END_IF
	IF AxisSetpointZ.Mapped THEN hrExtAxis := GetMostSignificant(hrExtAxis, AxisSetpointZ.Initialize());END_IF
	IF AxisSetpointA.Mapped THEN hrExtAxis := GetMostSignificant(hrExtAxis, AxisSetpointA.Initialize());END_IF
	IF AxisSetpointB.Mapped THEN hrExtAxis := GetMostSignificant(hrExtAxis, AxisSetpointB.Initialize());END_IF
	IF AxisSetpointC.Mapped THEN hrExtAxis := GetMostSignificant(hrExtAxis, AxisSetpointC.Initialize());END_IF
	
	bInitDone := (hrExtAxis = S_OK);	
	
	//Pending
	Initialize := S_PENDING;;	
ELSE	
	//Done
	Initialize := S_OK;	
END_IF


THIS^.fbFeedback.ActiveCommand 		:= TO_STRING(CHALET_NC.E_NcAxisCommands.Initialize);
THIS^.eActiveCommand 				:= CHALET_NC.E_NcAxisCommands.Initialize;
THIS^.fbFeedback.LastCommandAccepted:= TRUE;	
//Set done or keep in busy state	
THIS^.fbFeedback.HR := Initialize;
END_METHOD

{attribute 'monitoring':='call'}
PROPERTY Mapped : BOOL //Project is mapped to MC (McToPlc and PlcToMc)
GET
VAR
	bMcToPlcNotMapped 	: BOOL;
	bPlcToMcNotMapped 	: BOOL;
END_VAR
//F_GetMappingStatus is not working on IO Data Pointer
	//bPlcToMcNotMapped := F_GetMappingStatus(ADR(THIS^.fbMover.PlcToMc), SIZEOF(THIS^.fbMover.PlcToMc)) <> EPlcMappingStatus.MS_Mapped;
	//bMcToPlcNotMapped := F_GetMappingStatus(ADR(THIS^.fbMover.McToPlc), SIZEOF(THIS^.fbMover.McToPlc)) <> EPlcMappingStatus.MS_Mapped;

	
Mapped := THIS^.fbMover.MCTOPLC.STD.MoverOID <> 0;
END_GET
END_PROPERTY

{attribute 'monitoring':='call'}
PROPERTY Mode : MC_PLANAR_MOVER_COMMAND_MODE
GET
Mode := THIS^.fbMover.MCTOPLC.STD.CommandMode;
END_GET
END_PROPERTY

{attribute 'monitoring':='call'}
//Unique object ID
PROPERTY OID : OTCID
GET
OID := THIS^.fbMover.MCTOPLC.STD.MoverOID;
END_GET
END_PROPERTY

{attribute 'monitoring':='call'}
PROPERTY PlanarMover : REFERENCE TO MC_PlanarMover
GET
PlanarMover ref= THIS^.fbMover;
END_GET
END_PROPERTY

(* Time-critical information is processed here, which can then be polled via the property every cycle. 
The update method is usually at the end of the program and then it is already 'outdated'. *)
METHOD PRIVATE Prepare : HRESULT
VAR

END_VAR
VAR_INST
	{attribute 'hide'}
	nLastUpdatedCycleCount : UDINT;
END_VAR
//Check if this Cycle the dates are allready prepared
IF nLastUpdatedCycleCount <> TwinCAT_SystemInfoVarList._TaskInfo[THIS^.nTaskIndex].CycleCount THEN
	nLastUpdatedCycleCount := TwinCAT_SystemInfoVarList._TaskInfo[THIS^.nTaskIndex].CycleCount;

	

		
END_IF
END_METHOD

{attribute 'monitoring':='call'}
PROPERTY PUBLIC ProductData : I_XP_ProductData
GET
ProductData := ipProductData;
END_GET
SET
// No change. Same interface is set again
IF ipProductData = ProductData THEN
	;//Noting
	
ELSE

	// If allready an interface is linked. Unlink
	IF ipProductData <> 0 THEN
		ipProductData.LinkToMover(0);
		ipProductData := 0;
	END_IF
	
	// Link and store new interface
	IF ProductData <> 0 THEN
		ProductData.LinkToMover(THIS^);
		ipProductData := ProductData;
	END_IF
END_IF
END_SET
END_PROPERTY

{attribute 'monitoring':='call'}
PROPERTY Route : REFERENCE TO FB_CH_List
GET
Route ref= THIS^.fbRoute;
END_GET
END_PROPERTY

METHOD PUBLIC Update : HRESULT

// ********************** Set feedback depending on active command *******************************
IF THIS^.eActiveCommand <> E_NcAxisCommands.None THEN
	fbFeedback.ActiveCommand 	:= TO_STRING(THIS^.eActiveCommand);	
END_IF

CASE THIS^.eActiveCommand OF
	E_NcAxisCommands.None: 
		//Display if a Mover Error is active during no command is active
		IF THIS^.fbMover.Error AND NOT fbFeedback.Error THEN 
			IF THIS^.fbMover.ErrorId <> 1810(*ignore ADSERR_DEVICE_INVALIDSTATE*) THEN
				fbFeedback.ErrorId 			:= THIS^.fbMover.ErrorID;
				fbFeedback.ActiveCommand 	:= TO_STRING(E_NcAxisCommands.None);	
				fbFeedback.ClearObjectInfo();
			END_IF
		END_IF

	E_NcAxisCommands.Initialize:
		fbFeedback.Busy 			:= NOT THIS^.bInitDone;
		fbFeedback.Done 			:= THIS^.bInitDone;
		fbFeedback.ErrorId 			:= 0;
		fbFeedback.ClearObjectInfo();
		                        	
	E_NcAxisCommands.MoveA:     	
		fbFeedback.Busy 			:= fbFeedbackMoveA.Busy;
		fbFeedback.Done 			:= fbFeedbackMoveA.Done;
		fbFeedback.ErrorId 			:= fbFeedbackMoveA.ErrorID;
        fbFeedback.ObjectInfo		:= fbFeedbackMoveA.objectInfo;
                                	
	E_NcAxisCommands.MoveB:     	
		fbFeedback.Busy 			:= fbFeedbackMoveB.Busy;
		fbFeedback.Done 			:= fbFeedbackMoveB.Done;
		fbFeedback.ErrorId 			:= fbFeedbackMoveB.ErrorID;
        fbFeedback.ObjectInfo		:= fbFeedbackMoveB.objectInfo;
                                	
	E_NcAxisCommands.MoveC:     	
		fbFeedback.Busy 			:= fbFeedbackMoveC.Busy;
		fbFeedback.Done 			:= fbFeedbackMoveC.Done;
		fbFeedback.ErrorId 			:= fbFeedbackMoveC.ErrorID;
        fbFeedback.ObjectInfo		:= fbFeedbackMoveC.objectInfo;
                                	
	E_NcAxisCommands.MoveXY:    	
		fbFeedback.Busy 			:= fbFeedbackMoveXY.Busy;
		fbFeedback.Done 			:= fbFeedbackMoveXY.Done;
		fbFeedback.ErrorId 			:= fbFeedbackMoveXY.ErrorID;
        fbFeedback.ObjectInfo		:= fbFeedbackMoveXY.objectInfo;
                                	
	E_NcAxisCommands.MoveZ:     	
		fbFeedback.Busy 			:= fbFeedbackMoveZ.Busy;
		fbFeedback.Done 			:= fbFeedbackMoveZ.Done;
		fbFeedback.ErrorId 			:= fbFeedbackMoveZ.ErrorID;
        fbFeedback.ObjectInfo		:= fbFeedbackMoveZ.objectInfo;
                                	
	E_NcAxisCommands.Enable:    	
		fbFeedback.Busy 			:= fbFeedbackEnable.Busy;
		fbFeedback.Done 			:= fbFeedbackEnable.Done;
		fbFeedback.ErrorId 			:= fbFeedbackEnable.ErrorID;
        fbFeedback.ObjectInfo		:= fbFeedbackEnable.objectInfo;
                                	
	E_NcAxisCommands.Disable:   	
		fbFeedback.Busy 			:= fbFeedbackDisable.Busy;
		fbFeedback.Done 			:= fbFeedbackDisable.Done;
		fbFeedback.ErrorId 			:= fbFeedbackDisable.ErrorID;
        fbFeedback.ObjectInfo		:= fbFeedbackDisable.objectInfo;
                                	
	E_NcAxisCommands.Reset:     	
		fbFeedback.Busy 			:= fbFeedbackReset.Busy;
		fbFeedback.Done 			:= fbFeedbackReset.Done;
		fbFeedback.ErrorId 			:= fbFeedbackReset.ErrorID;
        fbFeedback.ObjectInfo		:= fbFeedbackReset.objectInfo;
                                	
	E_NcAxisCommands.Halt:      	
		fbFeedback.Busy 			:= fbFeedbackHalt.Busy;
		fbFeedback.Done 			:= fbFeedbackHalt.Done;
		fbFeedback.ErrorId 			:= fbFeedbackHalt.ErrorID;
        fbFeedback.ObjectInfo		:= fbFeedbackHalt.objectInfo;

	E_NcAxisCommands.AddToGroupe:
		fbFeedback.Busy 			:= fbFeedbackAddToGrp.Busy;
		fbFeedback.Done 			:= fbFeedbackAddToGrp.Done;
		fbFeedback.ErrorId 			:= fbFeedbackAddToGrp.ErrorID;
        fbFeedback.ObjectInfo		:= fbFeedbackAddToGrp.objectInfo;

	E_NcAxisCommands.RemoveFromGroupe:
		fbFeedback.Busy 			:= fbFeedbackRmvFromGrp.Busy;
		fbFeedback.Done 			:= fbFeedbackRmvFromGrp.Done;
		fbFeedback.ErrorId 			:= fbFeedbackRmvFromGrp.ErrorID;
        fbFeedback.ObjectInfo		:= fbFeedbackRmvFromGrp.objectInfo;
		
	E_NcAxisCommands.JoinTrack:
		fbFeedback.Busy 			:= fbFeedbackJoinTrack.Busy;
		fbFeedback.Done 			:= fbFeedbackJoinTrack.Done;
		fbFeedback.ErrorId 			:= fbFeedbackJoinTrack.ErrorID;
        fbFeedback.ObjectInfo		:= fbFeedbackJoinTrack.objectInfo;
		
	E_NcAxisCommands.MoveOnTrack:
		fbFeedback.Busy 			:= fbFeedbackMoveOnTrack.Busy;
		fbFeedback.Done 			:= fbFeedbackMoveOnTrack.Done;
		fbFeedback.ErrorId 			:= fbFeedbackMoveOnTrack.ErrorID;
        fbFeedback.ObjectInfo		:= fbFeedbackMoveOnTrack.objectInfo;
		
	
	//Add the 6 axis to the feedback			
	E_NcAxisCommands.StartExternalSetpoint:
 		fbFeedback.Busy 		:= fbFeedbackExtStart.Busy;
		fbFeedback.Done 		:= fbFeedbackExtStart.Done;
		fbFeedback.ErrorId 		:= fbFeedbackExtStart.ErrorID;
		fbFeedback.ClearObjectInfo();
		IF AxisSetpointX.Mapped THEN fbFeedback.HR := GetMostSignificant(fbFeedback.HR, AxisSetpointX.Feedback.HR);END_IF
		IF AxisSetpointY.Mapped THEN fbFeedback.HR := GetMostSignificant(fbFeedback.HR, AxisSetpointY.Feedback.HR);END_IF
		IF AxisSetpointZ.Mapped THEN fbFeedback.HR := GetMostSignificant(fbFeedback.HR, AxisSetpointZ.Feedback.HR);END_IF
		IF AxisSetpointA.Mapped THEN fbFeedback.HR := GetMostSignificant(fbFeedback.HR, AxisSetpointA.Feedback.HR);END_IF
		IF AxisSetpointB.Mapped THEN fbFeedback.HR := GetMostSignificant(fbFeedback.HR, AxisSetpointB.Feedback.HR);END_IF
		IF AxisSetpointC.Mapped THEN fbFeedback.HR := GetMostSignificant(fbFeedback.HR, AxisSetpointC.Feedback.HR);END_IF
		
	//Add the 6 axis to the feedback	
	E_NcAxisCommands.StopExternalSetpoint:
		fbFeedback.Busy 		:= fbFeedbackExtStop.Busy;
		fbFeedback.Done 		:= fbFeedbackExtStop.Done;
		fbFeedback.ErrorId 		:= fbFeedbackExtStop.ErrorID;
		fbFeedback.ClearObjectInfo(); 
		IF AxisSetpointX.Mapped THEN fbFeedback.HR := GetMostSignificant(fbFeedback.HR, AxisSetpointX.Feedback.HR);END_IF
		IF AxisSetpointY.Mapped THEN fbFeedback.HR := GetMostSignificant(fbFeedback.HR, AxisSetpointY.Feedback.HR);END_IF
		IF AxisSetpointZ.Mapped THEN fbFeedback.HR := GetMostSignificant(fbFeedback.HR, AxisSetpointZ.Feedback.HR);END_IF
		IF AxisSetpointA.Mapped THEN fbFeedback.HR := GetMostSignificant(fbFeedback.HR, AxisSetpointA.Feedback.HR);END_IF
		IF AxisSetpointB.Mapped THEN fbFeedback.HR := GetMostSignificant(fbFeedback.HR, AxisSetpointB.Feedback.HR);END_IF
		IF AxisSetpointC.Mapped THEN fbFeedback.HR := GetMostSignificant(fbFeedback.HR, AxisSetpointC.Feedback.HR);END_IF
		
		
	ELSE//External command in subclass
		;
END_CASE


// **********************  Stop to execute commands on .done or .error ***************************
IF fbFeedback.Done OR THIS^.fbFeedback.Error THEN
	eActiveCommand 				:= E_NcAxisCommands.None;
END_IF

//Update xplanar object
THIS^.fbMover.Update();
THIS^.UpdateExternalSetpoint();


//Update feedback object
fbFeedbackExtStart.Update(); 
fbFeedbackExtStop.Update(); 
fbFeedbackMoveA.Update(); 
fbFeedbackMoveB.Update(); 
fbFeedbackMoveC.Update(); 
fbFeedbackMoveXY.Update(); 
fbFeedbackMoveZ.Update(); 
fbFeedbackEnable.Update(); 
fbFeedbackDisable.Update(); 
fbFeedbackReset.Update(); 
fbFeedbackAddToGrp.Update(); 
fbFeedbackRmvFromGrp.Update(); 
fbFeedbackHalt.Update(); 
fbFeedbackJoinTrack.Update(); 
fbFeedbackMoveOnTrack.Update();
END_METHOD

END_FUNCTION_BLOCK

// COMPONENTs/Optional/Casting/ToXpTrack
FUNCTION ToXpTrack : BOOL
VAR_INPUT
	iChObject : I_CH_OBJECT;
	iXpTrack : REFERENCE TO I_XP_Track;
END_VAR

VAR
	iTmp : I_XP_Track;
END_VAR

(* 
   1. Test if the interface exists
   2. Test if the object implements a "Object" interface 
   3. Write reference to interface in parameter
   4. Returne TRUE if succesfull
*)
IF iChObject <> 0 AND_THEN __QUERYINTERFACE(iChObject,iTmp) THEN
	iXpTrack := iTmp;
	ToXpTrack := TRUE;
END_IF

END_FUNCTION

// COMPONENTs/Optional/Casting/ToXpMover
FUNCTION ToXpMover : BOOL
VAR_INPUT
	iChObject : I_CH_OBJECT;
	iXpMover : Reference to I_XP_Mover;
END_VAR

VAR
	iTmp : I_XP_Mover;
END_VAR

(* 
   1. Test if the interface exists
   2. Test if the object implements a "Object" interface 
   3. Write reference to interface in parameter
   4. Returne TRUE if succesfull
*)
IF iChObject <> 0 AND_THEN __QUERYINTERFACE(iChObject,iTmp) THEN
	iXpMover := iTmp;
	ToXpMover := TRUE;
END_IF

END_FUNCTION

// COMPONENTs/Optional/Casting/ToXpStation
FUNCTION ToXpStation : BOOL
VAR_INPUT
	iChObject : I_CH_OBJECT;
	iXpStation : REFERENCE TO I_XP_Station;
END_VAR

VAR
	iTmp : I_XP_Station;
END_VAR

(* Register the Station
   1. Test if the interface exists
   2. Test if the object implements a "Object" interface 
*)
IF iChObject <> 0 AND_THEN __QUERYINTERFACE(iChObject,iTmp) THEN
	iXpStation := iTmp;
	ToXpStation := TRUE;
END_IF

END_FUNCTION

// COMPONENTs/Optional/Trigger/FB_XP_Trigger
{attribute 'no_explicit_call' := 'Do not call the body - Stick to OOP'}
FUNCTION_BLOCK FB_XP_Trigger EXTENDS FB_CH_Object IMPLEMENTS I_XP_Trigger
VAR
	{attribute 'hide'}
	bInitDone : BOOL;
	{attribute 'hide'}
	ipXpSystem : I_XP_System_Registration;
	{attribute 'hide'}
	ipAccocietedTrack : I_XP_Track;
	{attribute 'hide'}
	ipListOfMoversToCheck : CHALET_BaseComponents.I_CH_LIST;
	{attribute 'hide'}
	fTriggerPositionOnTrack : LREAL;
	{attribute 'hide'}
	eTriggerDirection : Tc3_Mc3Definitions.MC_Direction := Tc3_Mc3Definitions.MC_DIRECTION.mcDirectionPositive;
	{attribute 'hide'}
	ipMoverAtTrigger : I_XP_Mover;
	{attribute 'hide'}
	aMoversPositionLastCycle : ARRAY [0..(CHALET_BaseComponents.BaseParameterlist.MAX_OBJECTS-1)] OF LREAL; // This list is generated at the end of the PRG and contais the positions. The positions are checked in the next cycle
	{attribute 'hide'}
	aMoversTrackLastCycle : ARRAY [0..(CHALET_BaseComponents.BaseParameterlist.MAX_OBJECTS-1)] OF I_XP_Track; // This list is generated at the end of the PRG and contais the track. The tracks are checked in the next cycle
	{attribute 'hide'}
	aMoversInterfaceLastCycle : ARRAY [0..(CHALET_BaseComponents.BaseParameterlist.MAX_OBJECTS-1)] OF I_XP_Mover; // This list is generated at the end of the PRG and contais the Mover interface. The positions are checked in the next cycle
END_VAR

{attribute 'monitoring':='call'}
PROPERTY AccocietedTrack : I_XP_Track
GET
AccocietedTrack := THIS^.ipAccocietedTrack;
END_GET
SET
THIS^.ipAccocietedTrack := AccocietedTrack;
END_SET
END_PROPERTY

METHOD FB_init : BOOL
VAR_INPUT
	bInitRetains : BOOL; // if TRUE, the retain variables are initialized (warm start / cold start)
	bInCopyCode : BOOL;  // if TRUE, the instance afterwards gets moved into the copy code (online change)
	
	ipXpSystem : I_XP_System_Registration; //Interface to XTS system object
	
END_VAR
VAR_INST
	{attribute 'hide'}
	bFBInitCalledOnce : BOOL; //Do the following code once during start up and not during onlinechange
END_VAR
//Do the following code once during start up and not during onlinechange
IF NOT bFBInitCalledOnce THEN 
	;
END_IF

//Regristrate object in System if unknown
IF ipXpSystem <> 0 AND THIS^.ipXpSystem = 0 THEN
	ipXpSystem.RegisterTrigger(THIS^);
	THIS^.ipXpSystem := ipXpSystem;
END_IF

bFBInitCalledOnce := TRUE;
END_METHOD

{attribute 'monitoring':='call'}
PROPERTY HR : HRESULT
GET
IF ipAccocietedTrack <> 0 AND_THEN ipAccocietedTrack.Length > 0 THEN
	HR := S_OK;
ELSE
	HR := E_FAIL;
END_IF
END_GET
END_PROPERTY

METHOD Initialize : HRESULT
IF THIS^.ipXpSystem = 0 THEN
	//No valide interface
	Initialize := E_FAIL;
	RETURN;
END_IF


THIS^.bInitDone := TRUE;
END_METHOD

PROPERTY ListOfMoversToCheck : I_CH_List
SET
IF ListOfMoversToCheck <> 0 THEN
	ipListOfMoversToCheck := ListOfMoversToCheck;
END_IF
END_SET
END_PROPERTY

{attribute 'monitoring':='call'}
PROPERTY MoverAtTrigger : I_XP_Mover
GET
THIS^.Prepare();//Prepare Time-critical information

MoverAtTrigger := ipMoverAtTrigger;
END_GET
END_PROPERTY

{attribute 'monitoring':='call'}
PROPERTY MoverDetected : BOOL
GET
THIS^.Prepare();//Prepare Time-critical information

MoverDetected := (ipMoverAtTrigger <> 0);
END_GET
END_PROPERTY

{attribute 'monitoring':='call'}
PROPERTY PositionOnTrack : LREAL
GET
PositionOnTrack := fTriggerPositionOnTrack;
END_GET
SET
fTriggerPositionOnTrack := PositionOnTrack;
END_SET
END_PROPERTY

(* Time-critical information is processed here, which can then be polled via the property every cycle. 
The update method is usually at the end of the program and then it is already 'outdated'. *)
METHOD PRIVATE Prepare : HRESULT
VAR
	fTrackLentgh : LREAL;
	fMoverActPos,fMoverLastPos : LREAL;
	ipMoverActTrack, ipMoverLastTrack : I_XP_Track;
	fRangePositive, fRangeNegative : LREAL;
	bTriggerIsCloseAtStartTrack, bTriggerIsCloseAtEndTrack : BOOL;
	bMoverWasInRangeNeg, bMoverWasInRangePos, bMoverIsInRangeNeg, bMoverIsInRangePos : BOOL;
	bMoverIsOnSameTrack, bMoverIsOnTrackAhead, bMoverIsOnTrackBehind, bMoverWasOnTrackAhead, bMoverWasOnTrackBehind : BOOL;
	nIdx, nIdxTrack : UDINT;
	fMaxMoveDistPerCycle : LREAL; //[mm] (2 m/s(max. xPlanar speed) * 20ms(max realistic SPS cycle time) + 10%)
END_VAR
VAR_INST
	{attribute 'hide'}
	nLastUpdatedCycleCount : UDINT;
END_VAR
VAR CONSTANT
END_VAR
IF NOT bInitDone OR (THIS^.ipListOfMoversToCheck = 0) OR (THIS^.ipAccocietedTrack = 0) THEN
	Prepare := E_FAIL;
	RETURN;
END_IF

//Check if this Cycle the dates are allready prepared
IF nLastUpdatedCycleCount <> TwinCAT_SystemInfoVarList._TaskInfo[THIS^.nTaskIndex].CycleCount THEN
	nLastUpdatedCycleCount := TwinCAT_SystemInfoVarList._TaskInfo[THIS^.nTaskIndex].CycleCount;
	
	//Abort on invalide interface - Get Track length
	IF ipAccocietedTrack = 0 THEN
		RETURN;
	END_IF
	fTrackLentgh := ipAccocietedTrack.Length;
	
	//Maximum distance a mover can travel in 1 plc cycle. Worstcase 2 m/s(max. xPlanar speed) * 20ms(max realistic SPS cycle time) + 10%
	fMaxMoveDistPerCycle := 2000.0(*2000mm/s=2mm/ms*) * (TwinCAT_SystemInfoVarList._TaskInfo[THIS^.nTaskIndex].CycleTime(*[100ns]*)/10_000)(*CycleTime ms*) / 1000.0 * 1.1(*10%*);
	
	//Clear last stored Mover if an new cycle has started
	THIS^.ipMoverAtTrigger := 0;
	
	//Check old list of Moverspositions and compare them to the current position of the same mover.
	//Set Trigger if the Mover pass the Station
	fRangePositive := MIN((THIS^.fTriggerPositionOnTrack + fMaxMoveDistPerCycle),fTrackLentgh);
	fRangeNegative := MAX((THIS^.fTriggerPositionOnTrack - fMaxMoveDistPerCycle),0); 
	bTriggerIsCloseAtStartTrack := (THIS^.fTriggerPositionOnTrack - fMaxMoveDistPerCycle) < 0.0;
	bTriggerIsCloseAtEndTrack 	:= (THIS^.fTriggerPositionOnTrack + fMaxMoveDistPerCycle) > fTrackLentgh;

		
	FOR nIdx := 0 TO (CHALET_BaseComponents.BaseParameterlist.MAX_OBJECTS-1) DO
		
		IF aMoversInterfaceLastCycle[nIdx] <> 0 THEN
			fMoverActPos 			:= aMoversInterfaceLastCycle[nIdx].PositionOnTrack;
			fMoverLastPos			:= aMoversPositionLastCycle[nIdx];
			ipMoverActTrack 		:= aMoversInterfaceLastCycle[nIdx].CurrentTrack;
			ipMoverLastTrack 		:= aMoversTrackLastCycle[nIdx];
			bMoverIsOnSameTrack 	:= (ipMoverActTrack = ipAccocietedTrack);
			
			//Abort if Lasttrack is not known. Example: first cycle after enabling
			IF ipMoverActTrack = 0 OR ipMoverLastTrack = 0 THEN
				RETURN;
			END_IF
			
			//Reset flags 
			bMoverIsOnTrackAhead 	:= FALSE;		bMoverIsOnTrackBehind 	:= FALSE;		bMoverWasOnTrackAhead 	:= FALSE;		bMoverWasOnTrackBehind 	:= FALSE;
			
			//Test all tracks before and after this track to recognize that the mover has just changed tracks. 
			//This is important if this trigger is near the end or beginning of a track
			FOR nIdxTrack := 0 TO (XPlanarParameterlist.N_MAX_STATIONS_AHEAD_OR_BEHIND-1) DO
				//Tracks Ahead - Mover Is/Was on Track ahead and close(cMaxMoveDistPerCycle) at beginn on track
				IF ipMoverActTrack.TracksStartFromThis[nIdxTrack] <> 0 THEN
					bMoverIsOnTrackAhead 	:= bMoverIsOnTrackAhead 	OR ((ipAccocietedTrack = ipMoverActTrack.TracksStartFromThis[nIdxTrack])  AND ((fMoverActPos - fMaxMoveDistPerCycle) < 0.0));
					bMoverWasOnTrackAhead 	:= bMoverWasOnTrackAhead 	OR ((ipAccocietedTrack = ipMoverLastTrack.TracksStartFromThis[nIdxTrack]) AND ((fMoverLastPos - fMaxMoveDistPerCycle) < 0.0));
				END_IF
				//Tracks Behind - Mover Is/Was on Track behind and close(cMaxMoveDistPerCycle) at end on track
				IF ipMoverActTrack.TracksEndAtThis[nIdxTrack] <> 0 THEN
					bMoverIsOnTrackBehind 	:= bMoverIsOnTrackBehind 	OR ((ipAccocietedTrack = ipMoverActTrack.TracksEndAtThis[nIdxTrack])  AND ((fMoverActPos	+ fMaxMoveDistPerCycle) > ipMoverActTrack.Length));
					bMoverWasOnTrackBehind 	:= bMoverWasOnTrackBehind 	OR ((ipAccocietedTrack = ipMoverLastTrack.TracksEndAtThis[nIdxTrack]) AND ((fMoverLastPos 	+ fMaxMoveDistPerCycle) > ipMoverLastTrack.Length));
				END_IF
			END_FOR
			
			//Closed track and station in close to Modulo pos
			IF bMoverIsOnSameTrack THEN
				bMoverIsOnTrackAhead 	:= ((fMoverActPos - fMaxMoveDistPerCycle) < 0.0);
				bMoverWasOnTrackAhead 	:= ((fMoverLastPos - fMaxMoveDistPerCycle) < 0.0);
				bMoverIsOnTrackBehind 	:= ((fMoverActPos	+ fMaxMoveDistPerCycle) > ipMoverActTrack.Length);
				bMoverWasOnTrackBehind 	:= ((fMoverLastPos 	+ fMaxMoveDistPerCycle) > ipMoverLastTrack.Length);
			END_IF
			
			//Check if Mover passes the station. Ex.: If the Trigger is at Pos 0mm on track, the Mover is never in bRangeNeg. For this case check for bMoverOnTrackBefore
			bMoverIsInRangePos 		:= ((fMoverActPos >= THIS^.fTriggerPositionOnTrack) AND (fMoverActPos <= fRangePositive) AND bMoverIsOnSameTrack) OR (bMoverIsOnTrackAhead 	 AND bTriggerIsCloseAtEndTrack);   
			bMoverIsInRangeNeg 		:= ((fMoverActPos <= THIS^.fTriggerPositionOnTrack) AND (fMoverActPos >= fRangeNegative) AND bMoverIsOnSameTrack) OR (bMoverIsOnTrackBehind  AND bTriggerIsCloseAtStartTrack);     
			bMoverWasInRangePos		:= ((fMoverLastPos > THIS^.fTriggerPositionOnTrack) AND (fMoverLastPos >= fRangeNegative) AND bMoverIsOnSameTrack) OR (bMoverWasOnTrackAhead  AND bTriggerIsCloseAtEndTrack);   
			bMoverWasInRangeNeg		:= ((fMoverLastPos < THIS^.fTriggerPositionOnTrack) AND (fMoverLastPos <= fRangePositive) AND bMoverIsOnSameTrack) OR (bMoverWasOnTrackBehind AND bTriggerIsCloseAtStartTrack);     			

			IF eTriggerDirection = Tc3_Mc3Definitions.MC_DIRECTION.mcDirectionPositive  AND bMoverWasInRangeNeg AND bMoverIsInRangePos AND NOT bMoverWasInRangePos THEN
				THIS^.ipMoverAtTrigger := aMoversInterfaceLastCycle[nIdx];
				RETURN;
			ELSIF eTriggerDirection = Tc3_Mc3Definitions.MC_DIRECTION.mcDirectionNegative AND bMoverIsInRangeNeg AND bMoverWasInRangePos AND NOT bMoverWasInRangeNeg THEN
				THIS^.ipMoverAtTrigger := aMoversInterfaceLastCycle[nIdx];
				RETURN;	
			END_IF
			
		END_IF
	END_FOR
END_IF
END_METHOD

{attribute 'monitoring':='call'}
PROPERTY TimeStamp : Tc2_EtherCAT.T_DCTIME64
GET
THIS^.Prepare();//Prepare Time-critical information

///zzz todo exact time stamp calculatioin
 IF ipMoverAtTrigger <> 0 THEN
	 TimeStamp := F_GetCurDcTaskTime64();
 ELSE
	 TimeStamp := 0;
 END_IF
END_GET
END_PROPERTY

{attribute 'monitoring':='call'}
PROPERTY TriggerDirection : Tc3_Mc3Definitions.MC_Direction
GET
TriggerDirection := eTriggerDirection;
END_GET
SET
IF TriggerDirection =Tc3_Mc3Definitions.MC_DIRECTION.mcDirectionPositive OR TriggerDirection = Tc3_Mc3Definitions.MC_DIRECTION.mcDirectionNegative THEN
	eTriggerDirection := TriggerDirection;
END_IF
END_SET
END_PROPERTY

METHOD Update : HRESULT
VAR
	nIndex : UINT;
	ipMover : I_XP_Mover;
END_VAR
//Force to do an init befor call update
IF NOT bInitDone THEN
	THIS^.Initialize();
	RETURN;
END_IF

//Clear array
MEMSET(destAddr:=ADR(aMoversInterfaceLastCycle),n:=SIZEOF(aMoversInterfaceLastCycle),fillByte:=0);
MEMSET(destAddr:=ADR(aMoversPositionLastCycle),n:=SIZEOF(aMoversPositionLastCycle),fillByte:=0);
MEMSET(destAddr:=ADR(aMoversTrackLastCycle),n:=SIZEOF(aMoversTrackLastCycle),fillByte:=0);

